(* CODESYS project Tc3_Mc3Ptp.library
   TcLibraryId: Beckhoff Automation GmbH|Tc3_Mc3Ptp|0.4.47.0
   Company: Beckhoff Automation GmbH
   Title: Tc3_Mc3Ptp
   Placeholder: Tc3_Mc3Ptp
   Version: 0.4.47.0

Project tree, tasks and I/O mapping:
  libraries: Tc3_Mc3Base, 0.4.47.0 (Beckhoff Automation GmbH)
  DUTs/
    function block AXIS_REF [ST]: FB_init, FB_exit, InitializeWithOid, GetMotionObjectOid, GetSetValue1DOid, GetActValue1DOid, Name, Oid
    data type AXIS_REF_TOMC
    data type AXIS_REF_TOPLC
    data type EJogMode
    data type EModuloDirection
    Enums/
      data type ELockingStrategy
      data type ETouchProbeSource
    data type EHomingMode
    data type ESource
    data type GearInLegacyOptions
    data type GearInOptions
    data type GearInPosOptions
    data type GearInPosLegacyOptions
    data type SetPositionOptions
    interface Type_ActValue1D: GetActValue1DOid
    interface Type_SetValue1D: GetSetValue1DOid
  POUs/
    Administrative/
      function block MC_Power [ST]: FB_init, FB_exit
      function block MC_SetOverride [ST]: FB_init, FB_exit
      function block MC_Reset [ST]: FB_init, FB_exit
      function block MC_ActivateExternalSetpointGeneration [ST]: FB_init, FB_exit
      function block MC_ReadActualPosition [ST]: FB_init, FB_exit
      function block MC_ReadAxisError [ST]: FB_init, FB_exit
      function block MC_ReadStatus [ST]: FB_init, FB_exit
      function block MC_SetPosition [ST]: FB_init, FB_exit
      function block MC_GetTimeAtActualPosition [ST]: FB_init, FB_exit
      function block MC_GetActualPositionAtTime [ST]: FB_init, FB_exit
      function block MC_TouchProbe [ST]: FB_init, FB_exit
      function block MC_TouchProbeContinuous [ST]: FB_init, FB_exit
      function block MC_AbortTrigger [ST]: FB_init, FB_exit
      function block MC_WriteHardwareParameterAsync [ST]: FB_init, FB_exit
      function block MC_ReadHardwareParameterAsync [ST]: FB_init, FB_exit
    Motion/
      function block MC_Halt [ST]: FB_init, FB_exit
      function block MC_GearIn [ST]: FB_init, FB_exit
      function block MC_GearInLegacy [ST]: FB_init, FB_exit
      function block MC_GearInPos [ST]: FB_init, FB_exit
      function block MC_GearInPosLegacy [ST]: FB_init, FB_exit
      function block MC_MoveAbsolute [ST]: FB_init, FB_exit
      function block MC_MoveModulo [ST]: FB_init, FB_exit
      function block MC_MoveRelative [ST]: FB_init, FB_exit
      function block MC_MoveVelocity [ST]: FB_init, FB_exit
      function block MC_Stop [ST]: FB_init, FB_exit
      function block MC_Home [ST]: FB_init, FB_exit
      function block MC_Jog [ST]: FB_init, FB_exit
      function block MC_WaitForStableActualPosition [ST]: FB_init, FB_exit
      function block MC_PhasingAbsolute [ST]: FB_init, FB_exit
      function block MC_PhasingRelative [ST]: FB_init, FB_exit
      function block MC_HaltPhasing [ST]: FB_init, FB_exit
  Version/
    global variables Global_Version
*)

// DUTs/AXIS_REF_TOMC
(* Contains the information of the AXIS_REF passed from PLC to MC. *)
{attribute 'TcIecLibraryType'}
{attribute 'Namespace' := 'Tc3_Mc3Ptp'}
TYPE AXIS_REF_TOMC : 
	STRUCT
		(* Standard data from PLC to MC. *)
		{attribute 'GUID' := '5A944F05-2D7C-4FD6-9ABA-134068F48E38'}
		{attribute 'Namespace' := 'MC'}
		Std : MC.CDT_PLCTOMC_AXIS_STD;
	END_STRUCT
END_TYPE

// DUTs/AXIS_REF_TOPLC
(* Contains the information of the AXIS_REF passed from PLC to MC. *)
{attribute 'TcIecLibraryType'}
{attribute 'Namespace' := 'Tc3_Mc3Ptp'}
TYPE AXIS_REF_TOPLC : 
	STRUCT
		(* Reference to standard data from MC to PLC. *)
		{attribute 'TcPointerMapping'}
		{attribute 'GUID' := '1FDF4C99-95D5-41A1-806D-90D273DC6BDC'}
		{attribute 'Namespace' := 'MC'}
		Std : REFERENCE TO MC.CDT_MCTOPLC_AXIS_STD;
		(* Reference to setpoint data from MC *)
		{attribute 'TcPointerMapping'}
		{attribute 'GUID' := '619A0C74-EA7E-46BA-B447-F4E8C97E41FB'}
		{attribute 'Namespace' := 'MC'}
		Set : REFERENCE TO MC.CDT_MCTOPLC_AXIS_SET;
		(* Reference to actpoint data from MC *)
		{attribute 'TcPointerMapping'}
		{attribute 'GUID' := 'A42D1F82-D46F-4C1C-8CEF-A7CF7DED130F'}
		{attribute 'Namespace' := 'MC'}
		Act : REFERENCE TO MC.CDT_MCTOPLC_AXIS_ACT;
		 {attribute 'hide'}
		_reserved1 : ARRAY [1..4] OF UINT_8_16;
		(* Reference to modulo positions of a modulo axis *)
		{attribute 'TcPointerMapping'}
		{attribute 'GUID' := 'D0D202B0-695B-4EBE-A25A-AE633C79AA06'}
		{attribute 'Namespace' := 'MC'}
		Modulo : REFERENCE TO MC.CDT_MCTOPLC_AXIS_MODULO;
		(* Reference to load data from MC *)
		{attribute 'TcPointerMapping'}
		{attribute 'GUID' := '222F7CA1-43FF-474A-AC84-1035F5DA7F7A'}
		{attribute 'Namespace' := 'MC'}
		Load : REFERENCE TO MC.CDT_MCTOPLC_AXIS_LOAD;
		 {attribute 'hide'}
		_reserved2 : ARRAY [1..8] OF UINT_8_16;
		(* Reference to fluidpower data from MC *)
		{attribute 'TcPointerMapping'}
		{attribute 'GUID' := 'FF85C83C-7A68-4103-B383-EFF835275DAB'}
		{attribute 'Namespace' := 'MC'}
		FluidPower : REFERENCE TO MC.CDT_MCTOPLC_AXIS_FLUIDPOWER;
	END_STRUCT
END_TYPE

// DUTs/EJogMode
{attribute 'TcIecLibraryType'}
{attribute 'Namespace' := 'Tc3_Mc3Ptp'}
{attribute 'strict'}
{attribute 'qualified_only'}
{attribute 'to_string'}
TYPE EJogMode : (StandardSlow:=1, StandardFast:=2, Continuous:=3, Inching:=4) UINT;
END_TYPE

// DUTs/EModuloDirection
{attribute 'TcIecLibraryType'}
{attribute 'Namespace' := 'Tc3_Mc3Ptp'}
{attribute 'strict'}
{attribute 'qualified_only'}
{attribute 'to_string'}
TYPE EModuloDirection : (ShortestDistance:=0, PositiveDirection:=1, NegativeDirection:=2) UINT;
END_TYPE

// DUTs/EHomingMode
{attribute 'TcIecLibraryType'}
{attribute 'Namespace' := 'Tc3_Mc3Ptp'}
{attribute 'qualified_only'}
{attribute 'strict'}
{attribute 'to_string'}
TYPE EHomingMode : (ForceIsPositionValid:=16#0, ResetIsPositionValid:=16#1, DirectSetPosition:=16#2) UDINT;
END_TYPE

// DUTs/ESource
{attribute 'TcIecLibraryType'}
{attribute 'Namespace' := 'Tc3_Mc3Ptp'}
{attribute 'hide'}
{attribute 'to_string'}
TYPE ESource : (SetValue:=0, ActualValue:=1) UINT;
END_TYPE

// DUTs/GearInLegacyOptions
(* Contains additional options for MC_GearInLegacy *)
{attribute 'TcIecLibraryType'}
{attribute 'Namespace' := 'Tc3_Mc3Ptp'}
{attribute 'hide'}
TYPE GearInLegacyOptions : 
	STRUCT
		{attribute 'Namespace' := 'Tc3_Mc3Base'}
		AllowedSlaveSyncDirections : Tc3_Mc3Base.ESyncDirection := Tc3_Mc3Base.ESyncDirection.Both;
		{attribute 'GUID' := 'AAA4D297-4BFA-4B3F-8507-5BB1F7885E81'}
		{attribute 'Namespace' := 'Tc3_Mc3Ptp'}
		LockingStrategy : ELockingStrategy := ELockingStrategy.PositionLocking;
	END_STRUCT
END_TYPE

// DUTs/GearInOptions
(* Contains additional options for MC_GearIn *)
{attribute 'TcIecLibraryType'}
{attribute 'Namespace' := 'Tc3_Mc3Ptp'}
{attribute 'hide'}
TYPE GearInOptions : 
	STRUCT
		HardcopyWhenInSync : BOOL := false;
	END_STRUCT
END_TYPE

// DUTs/GearInPosOptions
(* Contains additional options for MC_GearInPos *)
{attribute 'TcIecLibraryType'}
{attribute 'Namespace' := 'Tc3_Mc3Ptp'}
{attribute 'hide'}
TYPE GearInPosOptions : 
	STRUCT
		{attribute 'Namespace' := 'Tc3_Mc3Base'}
		AllowedSlaveSyncDirections : Tc3_Mc3Base.ESyncDirection := Tc3_Mc3Base.ESyncDirection.Both;
		 {attribute 'hide'}
		_reserved1 : UINT;
		(* Additional turns for this command *)
		AdditionalTurns : UDINT := 0;
		InSyncToleranceDistance : LREAL := 0;
	END_STRUCT
END_TYPE

// DUTs/GearInPosLegacyOptions
(* Contains additional options for MC_GearInPosLegacy *)
{attribute 'TcIecLibraryType'}
{attribute 'Namespace' := 'Tc3_Mc3Ptp'}
{attribute 'hide'}
TYPE GearInPosLegacyOptions : 
	STRUCT
		{attribute 'Namespace' := 'Tc3_Mc3Base'}
		AllowedSlaveSyncDirections : Tc3_Mc3Base.ESyncDirection := Tc3_Mc3Base.ESyncDirection.Both;
		 {attribute 'hide'}
		_reserved1 : ARRAY [1..6] OF USINT;
		InSyncToleranceDistance : LREAL := 0;
	END_STRUCT
END_TYPE

// DUTs/SetPositionOptions
(* Contains additional options for MC_SetPosition *)
{attribute 'TcIecLibraryType'}
{attribute 'Namespace' := 'Tc3_Mc3Ptp'}
TYPE SetPositionOptions : 
	STRUCT
		(* If TRUE, the position lag is cleared when the function block is executed. *)
		ClearPositionLag : BOOL := false;
	END_STRUCT
END_TYPE

// DUTs/Enums/ELockingStrategy
{attribute 'TcIecLibraryType'}
{attribute 'Namespace' := 'Tc3_Mc3Ptp'}
{attribute 'qualified_only'}
{attribute 'strict'}
{attribute 'to_string'}
TYPE ELockingStrategy : (VelocityLocking:=1, PositionLocking:=2) UINT := VelocityLocking;
END_TYPE

// DUTs/Enums/ETouchProbeSource
(* Selection for touch probe trigger input. *)
{attribute 'TcIecLibraryType'}
{attribute 'Namespace' := 'Tc3_Mc3Ptp'}
{attribute 'qualified_only'}
{attribute 'strict'}
{attribute 'to_string'}
TYPE ETouchProbeSource : (TouchProbe1:=1, TouchProbe2:=2, ExternalTrigger:=3) UINT;
END_TYPE

// Version/Global_Version
{attribute 'TcGenerated'}
// This function has been automatically generated from the project information.
VAR_GLOBAL CONSTANT
	{attribute 'const_non_replaced'}
	{attribute 'linkalways'}
	stLibVersion_Tc3_Mc3Ptp : ST_LibVersion := (iMajor := 0, iMinor := 4, iBuild := 47, iRevision := 0, nFlags := 0, sVersion := '0.4.47.0');
	{attribute 'const_non_replaced'}
	{attribute 'linkalways'}
	sLibraryId_Tc3_Mc3Ptp : String := 'Beckhoff Automation GmbH|Tc3_Mc3Ptp|0.4.47.0';
END_VAR

// DUTs/AXIS_REF

{attribute 'c++_compatible'}
{attribute 'external_name' := 'AXIS_REF_GUID_D3CA51BE_3DF9_1ECF_B7F2_294D2474676B'}
{attribute 'TcIecLibraryType'}
(* AXIS_REF data structure *)
FUNCTION_BLOCK AXIS_REF IMPLEMENTS Tc3_Mc3Base.Type_MotionObject, Type_SetValue1D, Type_ActValue1D
VAR
END_VAR
VAR_INPUT
	(* AXIS_REF outputs. *)
	{attribute 'GUID' := '90A3EB19-687D-4532-BDEE-19D8EA71F7B6'}
	{attribute 'Namespace' := 'Tc3_Mc3Ptp'}
	PlcToMc AT %Q* : AXIS_REF_TOMC;
	(* AXIS_REF inputs. *)
	{attribute 'GUID' := '6F07441C-203E-413F-A1C8-211D3A777892'}
	{attribute 'Namespace' := 'Tc3_Mc3Ptp'}
	McToPlc AT %I* : AXIS_REF_TOPLC;
END_VAR
VAR
	 {attribute 'hide'}
	_reserved1 : ARRAY [1..4] OF UINT_8_16;
END_VAR

{attribute 'TcTypeSystem'}

(* Internal method *)
{attribute 'hide'}
METHOD FB_init : BOOL
VAR_INPUT
	(*  if TRUE, the retain variables are initialized (warm start / cold start) *)
	bInitRetains : BOOL;
	(*  if TRUE, the instance afterwards gets moved into the copy code (online change) *)
	bInCopyCode : BOOL;
END_VAR
END_METHOD

{attribute 'TcTypeSystem'}

(* Internal method *)
{attribute 'hide'}
METHOD FB_exit : BOOL
VAR_INPUT
	(*  if TRUE, the exit method is called for exiting an instance that is copied afterwards (online change). *)
	bInCopyCode : BOOL;
END_VAR
END_METHOD

{attribute 'TcTypeSystem'}

(* Internal method to wrap OID *)
{attribute 'hide'}
METHOD InitializeWithOid
VAR_INPUT
	(*  Oid which is used as an alternative when this is used as master. *)
	{attribute 'GUID' := '18071995-0000-0000-0000-00000000000F'}
	NewOid : GLOBAL.OTCID;
END_VAR
END_METHOD

{attribute 'TcTypeSystem'}

{attribute 'c++_external'}
{attribute 'hide'}
METHOD GetMotionObjectOid : GLOBAL.OTCID
END_METHOD

{attribute 'TcTypeSystem'}

{attribute 'c++_external'}
{attribute 'hide'}
METHOD GetSetValue1DOid : GLOBAL.OTCID
END_METHOD

{attribute 'TcTypeSystem'}

{attribute 'c++_external'}
{attribute 'hide'}
METHOD GetActValue1DOid : GLOBAL.OTCID
END_METHOD

{attribute 'TcTypeSystem'}

{attribute 'monitoring' := 'call'}
	PROPERTY Name : STRING(255)
GET
END_GET
END_PROPERTY

{attribute 'TcTypeSystem'}

{attribute 'monitoring' := 'call'}
	PROPERTY Oid : GLOBAL.OTCID
GET
END_GET
END_PROPERTY

END_FUNCTION_BLOCK

// DUTs/Type_SetValue1D
{attribute 'Namespace' := 'Tc3_Mc3Ptp'}
{attribute 'c++_compatible'}
INTERFACE Type_SetValue1D

{attribute 'TcTypeSystem'}
{attribute 'c++_compatible'}
{attribute 'minimal_input_size' := '4'}
{attribute 'pack_mode' := '4'}
{attribute 'hide'}
METHOD GetSetValue1DOid : GLOBAL.OTCID
END_METHOD

END_INTERFACE

// DUTs/Type_ActValue1D
{attribute 'Namespace' := 'Tc3_Mc3Ptp'}
{attribute 'c++_compatible'}
INTERFACE Type_ActValue1D

{attribute 'TcTypeSystem'}
{attribute 'c++_compatible'}
{attribute 'minimal_input_size' := '4'}
{attribute 'pack_mode' := '4'}
{attribute 'hide'}
METHOD GetActValue1DOid : GLOBAL.OTCID
END_METHOD

END_INTERFACE

// POUs/Administrative/MC_Power

{attribute 'c++_compatible'}
{attribute 'external_name' := 'MC_Power_GUID_E3529116_274C_1460_937E_8AA859633871'}
{attribute 'TcIecLibraryType'}
{attribute 'hide_all_locals'}
(* 
		This function block controls the power stage (on or off).
	 *)
FUNCTION_BLOCK MC_Power
VAR_IN_OUT
	(* Reference to the axis *)
	{attribute 'GUID' := 'D3CA51BE-3DF9-1ECF-B7F2-294D2474676B'}
	{attribute 'Namespace' := 'Tc3_Mc3Ptp'}
	Axis : AXIS_REF;
END_VAR
VAR_INPUT
	(* General software enable for the axis *)
	Enable : BOOL;
	(* Feed enable in positive direction. Only effective if Enable = TRUE *)
	EnablePositive : BOOL := FALSE;
	(* Feed enable in negative direction. Only effective if Enable = TRUE *)
	EnableNegative : BOOL := FALSE;
END_VAR
VAR_OUTPUT
	(* Axis is operationally ready *)
	Status : BOOL;
	(* Axis has error *)
	Error : BOOL;
END_VAR
VAR
	 {attribute 'hide'}
	_reserved1 : ARRAY [1..3] OF USINT;
END_VAR
VAR_OUTPUT
	(* Axis error identifier *)
	ErrorId : UDINT;
END_VAR
VAR
	 {attribute 'hide'}
	_reserved2 : UINT_0_32;
END_VAR

{attribute 'TcTypeSystem'}

(* Internal method *)
{attribute 'hide'}
METHOD FB_init : BOOL
VAR_INPUT
	(*  if TRUE, the retain variables are initialized (warm start / cold start) *)
	bInitRetains : BOOL;
	(*  if TRUE, the instance afterwards gets moved into the copy code (online change) *)
	bInCopyCode : BOOL;
END_VAR
END_METHOD

{attribute 'TcTypeSystem'}

(* Internal method *)
{attribute 'hide'}
METHOD FB_exit : BOOL
VAR_INPUT
	(*  if TRUE, the exit method is called for exiting an instance that is copied afterwards (online change). *)
	bInCopyCode : BOOL;
END_VAR
END_METHOD

END_FUNCTION_BLOCK

// POUs/Administrative/MC_SetOverride

{attribute 'c++_compatible'}
{attribute 'external_name' := 'MC_SetOverride_GUID_121C7E78_08E0_1E5A_A94C_0DF92BBB78C9'}
{attribute 'TcIecLibraryType'}
{attribute 'hide_all_locals'}
(* 
	This function block sets the velocity override factor that is applied to movement commands of the axis.
	The override factor does not apply to movement in the synchronized motion state (e.g. movement induced by MC_GearIn, MC_GearInPos, ...).
	 *)
FUNCTION_BLOCK MC_SetOverride
VAR_IN_OUT
	(* Reference to the axis *)
	{attribute 'GUID' := 'D3CA51BE-3DF9-1ECF-B7F2-294D2474676B'}
	{attribute 'Namespace' := 'Tc3_Mc3Ptp'}
	Axis : AXIS_REF;
END_VAR
VAR_INPUT
	(* Write the velocity override factor continuously while Enable = TRUE *)
	Enable : BOOL;
END_VAR
VAR
	 {attribute 'hide'}
	_reserved1 : ARRAY [1..7] OF USINT;
END_VAR
VAR_INPUT
	(* Applies to commanded velocities. Valid range is [0,1]. Use STRING_TO_LREAL('#Ignore') to NOT overwrite the previous value. *)
	VelocityFactor : LREAL := 1.0;
END_VAR
VAR
	 {attribute 'hide'}
	_reserved2 : ARRAY [1..8] OF USINT;
END_VAR
VAR_OUTPUT
	(* The commanded override is set *)
	Enabled : BOOL;
	(* Error occurred within function block *)
	Error : BOOL;
END_VAR
VAR
	 {attribute 'hide'}
	_reserved3 : UINT;
END_VAR
VAR_OUTPUT
	(* Error identifier *)
	ErrorId : UDINT;
END_VAR

{attribute 'TcTypeSystem'}

(* Internal method *)
{attribute 'hide'}
METHOD FB_init : BOOL
VAR_INPUT
	(*  if TRUE, the retain variables are initialized (warm start / cold start) *)
	bInitRetains : BOOL;
	(*  if TRUE, the instance afterwards gets moved into the copy code (online change) *)
	bInCopyCode : BOOL;
END_VAR
END_METHOD

{attribute 'TcTypeSystem'}

(* Internal method *)
{attribute 'hide'}
METHOD FB_exit : BOOL
VAR_INPUT
	(*  if TRUE, the exit method is called for exiting an instance that is copied afterwards (online change). *)
	bInCopyCode : BOOL;
END_VAR
END_METHOD

END_FUNCTION_BLOCK

// POUs/Motion/MC_GearIn

{attribute 'c++_compatible'}
{attribute 'external_name' := 'MC_GearIn_GUID_E9493D77_974B_13E8_841A_4F997893F8D6'}
{attribute 'TcIecLibraryType'}
{attribute 'hide_all_locals'}
{attribute 'hide'}
(* 
		This function block commands a ratio between the velocity of the slave and master axis.
	 *)
FUNCTION_BLOCK MC_GearIn
VAR_INPUT
	(* Reference to the master axis *)
	{attribute 'GUID' := '67A81BB4-B31C-4E6F-99E0-6B37521E2266'}
	{attribute 'Namespace' := 'Tc3_Mc3Ptp'}
	Master : Type_ActValue1D;
	(* Reference to the slave axis *)
	{attribute 'GUID' := '71DDD02B-B842-4DDB-8CBB-D377B6714EDA'}
	{attribute 'Namespace' := 'Tc3_Mc3Ptp'}
	Slave : Type_SetValue1D;
	(* Trigger the command with rising edge *)
	Execute : BOOL;
END_VAR
VAR
	 {attribute 'hide'}
	_reserved1 : UINT_24_56;
END_VAR
VAR_INPUT
	(* Gear ratio numerator *)
	RatioNumerator : LREAL := 1.0;
	(* Gear ratio denominator *)
	RatioDenominator : UDINT := 1;
END_VAR
VAR
	 {attribute 'hide'}
	_reserved2 : UDINT;
END_VAR
VAR_INPUT
	(* Maximum slave velocity ([PosUnit]/s, positive) *)
	Velocity : LREAL := STRING_TO_LREAL('#Maximum');
	(* Maximum slave acceleration ([PosUnit]/s^2, positive) *)
	Acceleration : LREAL := STRING_TO_LREAL('#Default');
	(* Maximum slave deceleration ([PosUnit]/s^2, positive) *)
	Deceleration : LREAL := STRING_TO_LREAL('#Default');
	(* Maximum slave jerk ([PosUnit]/s^3, positive) *)
	Jerk : LREAL := STRING_TO_LREAL('#Default');
	(* Chronological sequence of the command *)
	{attribute 'Namespace' := 'Tc3_Mc3Base'}
	BufferMode : Tc3_Mc3Base.EBufferMode := Tc3_Mc3Base.EBufferMode.Aborting;
	(* Reaction if an error occurs in the master while this command is active *)
	{attribute 'Namespace' := 'Tc3_Mc3Base'}
	ReactionToMasterError : Tc3_Mc3Base.EReactionToMasterError := Tc3_Mc3Base.EReactionToMasterError.TriggerSlaveError;
	(* Reaction if an error occurs in the slave while this command is active *)
	{attribute 'Namespace' := 'Tc3_Mc3Base'}
	ReactionToSlaveError : Tc3_Mc3Base.EReactionToSlaveError := Tc3_Mc3Base.EReactionToSlaveError.TriggerMasterError;
	(* Advanced function block options *)
	{attribute 'hide'}
	{attribute 'GUID' := 'BA63A6CC-1764-4B99-91C8-CC6CC375B652'}
	{attribute 'Namespace' := 'Tc3_Mc3Ptp'}
	Options : GearInOptions;
END_VAR
VAR_OUTPUT
	(* Synchronization established *)
	InGear : BOOL;
	(* Function block is not finished and new output values are to be expected *)
	Busy : BOOL;
	(* Function block has active control on the axis *)
	Active : BOOL;
	(* Command is aborted by another command *)
	CommandAborted : BOOL;
	(* Error occurred within function block *)
	Error : BOOL;
	(* Error identifier *)
	ErrorId : UDINT;
	(* Master is in error state *)
	MasterHasError : BOOL;
END_VAR
VAR
	 {attribute 'hide'}
	_reserved3 : UINT_24_56;
	 {attribute 'hide'}
	_reserved4 : ARRAY [1..28] OF UINT_8_16;
	 {attribute 'hide'}
	_reserved5 : ARRAY [1..32] OF USINT;
END_VAR

{attribute 'TcTypeSystem'}

(* Internal method *)
{attribute 'hide'}
METHOD FB_init : BOOL
VAR_INPUT
	(*  if TRUE, the retain variables are initialized (warm start / cold start) *)
	bInitRetains : BOOL;
	(*  if TRUE, the instance afterwards gets moved into the copy code (online change) *)
	bInCopyCode : BOOL;
END_VAR
END_METHOD

{attribute 'TcTypeSystem'}

(* Internal method *)
{attribute 'hide'}
METHOD FB_exit : BOOL
VAR_INPUT
	(*  if TRUE, the exit method is called for exiting an instance that is copied afterwards (online change). *)
	bInCopyCode : BOOL;
END_VAR
END_METHOD

END_FUNCTION_BLOCK

// POUs/Motion/MC_GearInPos

{attribute 'c++_compatible'}
{attribute 'external_name' := 'MC_GearInPos_GUID_B2BB4DF7_3ADC_10B7_8213_E2CF5BFD21E3'}
{attribute 'TcIecLibraryType'}
{attribute 'hide_all_locals'}
{attribute 'hide'}
(* 
		This function block commands a gear ratio between the position of the slave and master axes
		from the synchronization point onwards.
	 *)
FUNCTION_BLOCK MC_GearInPos
VAR_INPUT
	(* Reference to the master axis *)
	{attribute 'GUID' := '67A81BB4-B31C-4E6F-99E0-6B37521E2266'}
	{attribute 'Namespace' := 'Tc3_Mc3Ptp'}
	Master : Type_ActValue1D;
	(* Reference to the slave axis *)
	{attribute 'GUID' := '71DDD02B-B842-4DDB-8CBB-D377B6714EDA'}
	{attribute 'Namespace' := 'Tc3_Mc3Ptp'}
	Slave : Type_SetValue1D;
	(* Trigger the command with rising edge *)
	Execute : BOOL;
END_VAR
VAR
	 {attribute 'hide'}
	_reserved1 : UINT_24_56;
END_VAR
VAR_INPUT
	(* Gear ratio numerator *)
	RatioNumerator : LREAL := 1.0;
	(* Gear ratio denominator *)
	RatioDenominator : UDINT := 1;
END_VAR
VAR
	 {attribute 'hide'}
	_reserved2 : UDINT;
END_VAR
VAR_INPUT
	(* Position of master axis where master and slave axis are synchronized *)
	MasterSyncPosition : LREAL := STRING_TO_LREAL('#Invalid');
	(* Position of slave axis where master and slave axis are synchronized *)
	SlaveSyncPosition : LREAL := STRING_TO_LREAL('#Invalid');
	(* Maximum velocity during synchronization ([PosUnit]/s, positive) *)
	Velocity : LREAL := STRING_TO_LREAL('#Maximum');
	(* Maximum acceleration during synchronization ([PosUnit]/s^2, positive) *)
	Acceleration : LREAL := STRING_TO_LREAL('#Default');
	(* Maximum deceleration during synchronization ([PosUnit]/s^2, positive) *)
	Deceleration : LREAL := STRING_TO_LREAL('#Default');
	(* Maximum jerk during synchronization ([PosUnit]/s^3, positive) *)
	Jerk : LREAL := STRING_TO_LREAL('#Default');
	(* Chronological sequence of the command *)
	{attribute 'Namespace' := 'Tc3_Mc3Base'}
	BufferMode : Tc3_Mc3Base.EBufferMode := Tc3_Mc3Base.EBufferMode.Aborting;
	(* Reaction if an error occurs in the master while this command is active *)
	{attribute 'Namespace' := 'Tc3_Mc3Base'}
	ReactionToMasterError : Tc3_Mc3Base.EReactionToMasterError := Tc3_Mc3Base.EReactionToMasterError.TriggerSlaveError;
	(* Reaction if an error occurs in the slave while this command is active *)
	{attribute 'Namespace' := 'Tc3_Mc3Base'}
	ReactionToSlaveError : Tc3_Mc3Base.EReactionToSlaveError := Tc3_Mc3Base.EReactionToSlaveError.TriggerMasterError;
END_VAR
VAR
	 {attribute 'hide'}
	_reserved3 : UINT;
END_VAR
VAR_INPUT
	(* Advanced function block options *)
	{attribute 'hide'}
	{attribute 'GUID' := 'EB67571F-2653-4A23-A3F5-C429B6BFB18A'}
	{attribute 'Namespace' := 'Tc3_Mc3Ptp'}
	Options : GearInPosOptions;
END_VAR
VAR_OUTPUT
	(* Synchronization started *)
	{attribute 'hide'}
	StartSync : BOOL;
	(* Synchronization established *)
	InSync : BOOL;
	(* Function block is not finished and new output values are to be expected *)
	Busy : BOOL;
	(* Function block has active control on the axis *)
	Active : BOOL;
	(* Command is aborted by another command *)
	CommandAborted : BOOL;
	(* Error occurred within function block *)
	Error : BOOL;
END_VAR
VAR
	 {attribute 'hide'}
	_reserved4 : UINT;
END_VAR
VAR_OUTPUT
	(* Error identifier *)
	ErrorId : UDINT;
	(* Master is in error state *)
	MasterHasError : BOOL;
END_VAR
VAR
	 {attribute 'hide'}
	_reserved5 : UINT_24_56;
	 {attribute 'hide'}
	_reserved6 : ARRAY [1..28] OF UINT_8_16;
	 {attribute 'hide'}
	_reserved7 : ARRAY [1..28] OF USINT;
END_VAR

{attribute 'TcTypeSystem'}

(* Internal method *)
{attribute 'hide'}
METHOD FB_init : BOOL
VAR_INPUT
	(*  if TRUE, the retain variables are initialized (warm start / cold start) *)
	bInitRetains : BOOL;
	(*  if TRUE, the instance afterwards gets moved into the copy code (online change) *)
	bInCopyCode : BOOL;
END_VAR
END_METHOD

{attribute 'TcTypeSystem'}

(* Internal method *)
{attribute 'hide'}
METHOD FB_exit : BOOL
VAR_INPUT
	(*  if TRUE, the exit method is called for exiting an instance that is copied afterwards (online change). *)
	bInCopyCode : BOOL;
END_VAR
END_METHOD

END_FUNCTION_BLOCK

// POUs/Administrative/MC_Reset

{attribute 'c++_compatible'}
{attribute 'external_name' := 'MC_Reset_GUID_394AFEA2_BA6F_1DD1_8FD5_98DB85D7F990'}
{attribute 'TcIecLibraryType'}
{attribute 'hide_all_locals'}
(* 
		This function block resets all axis-related errors and transitions the axis out of state ErrorStop.<br/>
		The resulting state is Disabled, if no Enable is requested for the axis (e.g. via MC_Power).<br/>
		It results in DiscreteMotion, if the axis has a closed control loop and a controlled error reaction is still ongoing.<br/>
		Otherwise, standstill is the resultig state. This function block does not affect the output of motion function block instances.
	 *)
FUNCTION_BLOCK MC_Reset
VAR_INPUT
	(* Reference to the axis *)
	{attribute 'Namespace' := 'Tc3_Mc3Base'}
	Axis : Tc3_Mc3Base.Type_MotionObject;
	(* Trigger the command with rising edge *)
	Execute : BOOL;
END_VAR
VAR_OUTPUT
	(* Standstill state is reached *)
	Done : BOOL;
	(* Function block is not finished and new output values are to be expected *)
	Busy : BOOL;
	(* Error occurred within function block *)
	Error : BOOL;
	(* Error identifier *)
	ErrorId : UDINT;
END_VAR
VAR
	 {attribute 'hide'}
	_reserved1 : UINT_0_32;
	 {attribute 'hide'}
	_reserved2 : ARRAY [1..20] OF UINT_8_16;
	 {attribute 'hide'}
	_reserved3 : ARRAY [1..28] OF USINT;
END_VAR

{attribute 'TcTypeSystem'}

(* Internal method *)
{attribute 'hide'}
METHOD FB_init : BOOL
VAR_INPUT
	(*  if TRUE, the retain variables are initialized (warm start / cold start) *)
	bInitRetains : BOOL;
	(*  if TRUE, the instance afterwards gets moved into the copy code (online change) *)
	bInCopyCode : BOOL;
END_VAR
END_METHOD

{attribute 'TcTypeSystem'}

(* Internal method *)
{attribute 'hide'}
METHOD FB_exit : BOOL
VAR_INPUT
	(*  if TRUE, the exit method is called for exiting an instance that is copied afterwards (online change). *)
	bInCopyCode : BOOL;
END_VAR
END_METHOD

END_FUNCTION_BLOCK

// POUs/Administrative/MC_ActivateExternalSetpointGeneration

{attribute 'c++_compatible'}
{attribute 'external_name' := 'MC_ActivateExternalSetpointGeneration_GUID_3255B2A5_BCDE_1F3F_B215_3D486370678C'}
{attribute 'TcIecLibraryType'}
{attribute 'hide_all_locals'}
(* 
		This function block activates external setpoint generation. 
		Setpoints are generated by a function block, which is called through the ITcMcExternalSetpointGenerator interface from the MC context.
		Additionally custom startup data can be passed through the generator.
	 *)
FUNCTION_BLOCK MC_ActivateExternalSetpointGeneration
VAR_INPUT
	(* Reference to the axis *)
	{attribute 'GUID' := '71DDD02B-B842-4DDB-8CBB-D377B6714EDA'}
	{attribute 'Namespace' := 'Tc3_Mc3Ptp'}
	Axis : Type_SetValue1D;
	(* Trigger the command with rising edge *)
	Execute : BOOL;
END_VAR
VAR
	 {attribute 'hide'}
	_reserved1 : UINT_24_56;
END_VAR
VAR_INPUT
	(* External setpoint generator function block *)
	{attribute 'GUID' := 'EF828E0B-69F0-4553-9DFF-4817D2FD6510'}
	ExternalSetpointGenerator : GLOBAL.ITcMcExternalSetpointGenerator;
	(* (reserved) *)
	AllowOtherContext : BOOL := FALSE;
	(* Trigger error on inconsistent setpoint values (position, velocity, acceleration) if EnableDynamicChecks = TRUE *)
	EnableDynamicChecks : BOOL := TRUE;
END_VAR
VAR
	 {attribute 'hide'}
	_reserved2 : UINT_16_48;
END_VAR
VAR_INPUT
	(* Invocation identifier. The InvokeId can be used to identify an external setpoint generator in case external 
		setpoint generation is activated multiple times with the same ExternalSetpointGenerator. Another possibility is to transfer 
		custom data (for example a pointer to data struct) by this InvokeId. *)
	{attribute 'GUID' := '18071995-0000-0000-0000-000000000073'}
	{attribute 'GlobalType'}
	InvokeId : GLOBAL.XWORD := 0;
	(* Chronological sequence of the command *)
	{attribute 'Namespace' := 'Tc3_Mc3Base'}
	BufferMode : Tc3_Mc3Base.EBufferMode := Tc3_Mc3Base.EBufferMode.Aborting;
END_VAR
VAR_OUTPUT
	(* Function block is not finished and new output values are to be expected *)
	Busy : BOOL;
	(* Function block has active control on the axis *)
	Active : BOOL;
	(* Command is aborted by another command *)
	CommandAborted : BOOL;
	(* Error occurred within function block *)
	Error : BOOL;
END_VAR
VAR
	 {attribute 'hide'}
	_reserved3 : UINT;
END_VAR
VAR_OUTPUT
	(* Error identifier *)
	ErrorId : UDINT;
END_VAR
VAR
	 {attribute 'hide'}
	_reserved4 : UINT_0_32;
	 {attribute 'hide'}
	_reserved5 : ARRAY [1..32] OF UINT_8_16;
	 {attribute 'hide'}
	_reserved6 : ARRAY [1..24] OF USINT;
END_VAR

{attribute 'TcTypeSystem'}

(* Internal method *)
{attribute 'hide'}
METHOD FB_init : BOOL
VAR_INPUT
	(*  if TRUE, the retain variables are initialized (warm start / cold start) *)
	bInitRetains : BOOL;
	(*  if TRUE, the instance afterwards gets moved into the copy code (online change) *)
	bInCopyCode : BOOL;
END_VAR
END_METHOD

{attribute 'TcTypeSystem'}

(* Internal method *)
{attribute 'hide'}
METHOD FB_exit : BOOL
VAR_INPUT
	(*  if TRUE, the exit method is called for exiting an instance that is copied afterwards (online change). *)
	bInCopyCode : BOOL;
END_VAR
END_METHOD

END_FUNCTION_BLOCK

// POUs/Administrative/MC_ReadActualPosition

{attribute 'c++_compatible'}
{attribute 'external_name' := 'MC_ReadActualPosition_GUID_3C39B8D5_BF98_1B0D_873D_11943FFCDFE9'}
{attribute 'TcIecLibraryType'}
{attribute 'hide_all_locals'}
{attribute 'hide'}
(* 
		This function block reads the current axis actual position.
	 *)
FUNCTION_BLOCK MC_ReadActualPosition
VAR_IN_OUT
	(* Reference to the axis *)
	{attribute 'GUID' := 'D3CA51BE-3DF9-1ECF-B7F2-294D2474676B'}
	{attribute 'Namespace' := 'Tc3_Mc3Ptp'}
	Axis : AXIS_REF;
END_VAR
VAR_INPUT
	(* Read the actual position continuously while Enable = TRUE *)
	Enable : BOOL;
END_VAR
VAR_OUTPUT
	(* Valid output available at function block *)
	Valid : BOOL;
	(* Function block is not finished and new output values are to be expected *)
	Busy : BOOL;
	(* Error occurred within function block *)
	Error : BOOL;
	(* Error identifier *)
	ErrorId : UDINT;
	(* Actual position ([PosUnit]) *)
	Position : LREAL;
END_VAR

{attribute 'TcTypeSystem'}

(* Internal method *)
{attribute 'hide'}
METHOD FB_init : BOOL
VAR_INPUT
	(*  if TRUE, the retain variables are initialized (warm start / cold start) *)
	bInitRetains : BOOL;
	(*  if TRUE, the instance afterwards gets moved into the copy code (online change) *)
	bInCopyCode : BOOL;
END_VAR
END_METHOD

{attribute 'TcTypeSystem'}

(* Internal method *)
{attribute 'hide'}
METHOD FB_exit : BOOL
VAR_INPUT
	(*  if TRUE, the exit method is called for exiting an instance that is copied afterwards (online change). *)
	bInCopyCode : BOOL;
END_VAR
END_METHOD

END_FUNCTION_BLOCK

// POUs/Administrative/MC_ReadAxisError

{attribute 'c++_compatible'}
{attribute 'external_name' := 'MC_ReadAxisError_GUID_C6F572C1_61AE_1DA6_A376_F0A2AD8A74DD'}
{attribute 'TcIecLibraryType'}
{attribute 'hide_all_locals'}
{attribute 'hide'}
(* 
		This function block reads the current axis error identifier.
	 *)
FUNCTION_BLOCK MC_ReadAxisError
VAR_IN_OUT
	(* Reference to the axis *)
	{attribute 'GUID' := 'D3CA51BE-3DF9-1ECF-B7F2-294D2474676B'}
	{attribute 'Namespace' := 'Tc3_Mc3Ptp'}
	Axis : AXIS_REF;
END_VAR
VAR_INPUT
	(* Read the axis error identifier continuously while Enable = TRUE *)
	Enable : BOOL;
END_VAR
VAR_OUTPUT
	(* Valid output available at function block *)
	Valid : BOOL;
	(* Function block is not finished and new output values are to be expected *)
	Busy : BOOL;
	(* Error occurred within function block *)
	Error : BOOL;
	(* Error identifier *)
	ErrorId : UDINT;
	(* Axis error identifier *)
	AxisErrorId : UDINT;
END_VAR
VAR
	 {attribute 'hide'}
	_reserved1 : UINT_0_32;
END_VAR

{attribute 'TcTypeSystem'}

(* Internal method *)
{attribute 'hide'}
METHOD FB_init : BOOL
VAR_INPUT
	(*  if TRUE, the retain variables are initialized (warm start / cold start) *)
	bInitRetains : BOOL;
	(*  if TRUE, the instance afterwards gets moved into the copy code (online change) *)
	bInCopyCode : BOOL;
END_VAR
END_METHOD

{attribute 'TcTypeSystem'}

(* Internal method *)
{attribute 'hide'}
METHOD FB_exit : BOOL
VAR_INPUT
	(*  if TRUE, the exit method is called for exiting an instance that is copied afterwards (online change). *)
	bInCopyCode : BOOL;
END_VAR
END_METHOD

END_FUNCTION_BLOCK

// POUs/Administrative/MC_ReadStatus

{attribute 'c++_compatible'}
{attribute 'external_name' := 'MC_ReadStatus_GUID_294643E2_96D8_11B0_8DA0_D7A71A4F8120'}
{attribute 'TcIecLibraryType'}
{attribute 'hide_all_locals'}
(* 
		This function block reads the current axis state.
	 *)
FUNCTION_BLOCK MC_ReadStatus
VAR_IN_OUT
	(* Reference to the axis *)
	{attribute 'GUID' := 'D3CA51BE-3DF9-1ECF-B7F2-294D2474676B'}
	{attribute 'Namespace' := 'Tc3_Mc3Ptp'}
	Axis : AXIS_REF;
END_VAR
VAR_INPUT
	(* Read the axis state continuously while Enable = TRUE *)
	Enable : BOOL;
END_VAR
VAR_OUTPUT
	(* Valid output available at function block *)
	Valid : BOOL;
	(* Error occurred within function block *)
	Error : BOOL;
END_VAR
VAR
	 {attribute 'hide'}
	_reserved1 : USINT;
END_VAR
VAR_OUTPUT
	(* Error identifier *)
	ErrorId : UDINT;
	(* Axis is in state ErrorStop *)
	ErrorStop : BOOL;
	(* Axis is in state Disabled *)
	Disabled : BOOL;
	(* Axis is in state Stopping *)
	Stopping : BOOL;
	(* Axis is in state Homing *)
	Homing : BOOL;
	(* Axis is in state Standstill *)
	Standstill : BOOL;
	(* Axis is in state DiscreteMotion *)
	DiscreteMotion : BOOL;
	(* Axis is in state ContinuousMotion *)
	ContinuousMotion : BOOL;
	(* Axis is in state SynchronizedMotion *)
	SynchronizedMotion : BOOL;
END_VAR

{attribute 'TcTypeSystem'}

(* Internal method *)
{attribute 'hide'}
METHOD FB_init : BOOL
VAR_INPUT
	(*  if TRUE, the retain variables are initialized (warm start / cold start) *)
	bInitRetains : BOOL;
	(*  if TRUE, the instance afterwards gets moved into the copy code (online change) *)
	bInCopyCode : BOOL;
END_VAR
END_METHOD

{attribute 'TcTypeSystem'}

(* Internal method *)
{attribute 'hide'}
METHOD FB_exit : BOOL
VAR_INPUT
	(*  if TRUE, the exit method is called for exiting an instance that is copied afterwards (online change). *)
	bInCopyCode : BOOL;
END_VAR
END_METHOD

END_FUNCTION_BLOCK

// POUs/Administrative/MC_SetPosition

{attribute 'c++_compatible'}
{attribute 'external_name' := 'MC_SetPosition_GUID_75691C58_C510_1BCF_81F5_23E77C57D1A7'}
{attribute 'TcIecLibraryType'}
{attribute 'hide_all_locals'}
(* 
		This function block shifts the coordinate system of an axis by manipulating both the setpoint position as well as the
		actual position of an axis with the same value without any movement caused (Re-calibration with same following error).
		This can be used for instance for a reference situation.
	 *)
FUNCTION_BLOCK MC_SetPosition
VAR_INPUT
	(* Reference to the axis *)
	{attribute 'GUID' := '71DDD02B-B842-4DDB-8CBB-D377B6714EDA'}
	{attribute 'Namespace' := 'Tc3_Mc3Ptp'}
	Axis : Type_SetValue1D;
	(* Trigger the command with rising edge *)
	Execute : BOOL;
END_VAR
VAR
	 {attribute 'hide'}
	_reserved1 : ARRAY [1..7] OF USINT;
END_VAR
VAR_INPUT
	(* New position value ([PosUnit]) or distance if Relative = TRUE *)
	Position : LREAL := STRING_TO_LREAL('#Invalid');
	(* Shift axis position by value *)
	Relative : BOOL := FALSE;
	(* Advanced function block options *)
	{attribute 'GUID' := '8BDBC654-D053-42BE-BD59-268374CF5136'}
	{attribute 'Namespace' := 'Tc3_Mc3Ptp'}
	Options : SetPositionOptions;
END_VAR
VAR_OUTPUT
	(* Position has new value *)
	Done : BOOL;
	(* Function block is not finished and new output values are to be expected *)
	Busy : BOOL;
	(* Error occurred within function block *)
	Error : BOOL;
END_VAR
VAR
	 {attribute 'hide'}
	_reserved2 : ARRAY [1..3] OF USINT;
END_VAR
VAR_OUTPUT
	(* Error identifier *)
	ErrorId : UDINT;
END_VAR
VAR
	 {attribute 'hide'}
	_reserved3 : UINT_0_32;
	 {attribute 'hide'}
	_reserved4 : ARRAY [1..20] OF UINT_8_16;
	 {attribute 'hide'}
	_reserved5 : ARRAY [1..32] OF USINT;
END_VAR

{attribute 'TcTypeSystem'}

(* Internal method *)
{attribute 'hide'}
METHOD FB_init : BOOL
VAR_INPUT
	(*  if TRUE, the retain variables are initialized (warm start / cold start) *)
	bInitRetains : BOOL;
	(*  if TRUE, the instance afterwards gets moved into the copy code (online change) *)
	bInCopyCode : BOOL;
END_VAR
END_METHOD

{attribute 'TcTypeSystem'}

(* Internal method *)
{attribute 'hide'}
METHOD FB_exit : BOOL
VAR_INPUT
	(*  if TRUE, the exit method is called for exiting an instance that is copied afterwards (online change). *)
	bInCopyCode : BOOL;
END_VAR
END_METHOD

END_FUNCTION_BLOCK

// POUs/Administrative/MC_GetTimeAtActualPosition

{attribute 'c++_compatible'}
{attribute 'external_name' := 'MC_GetTimeAtActualPosition_GUID_0CA0D808_4FD4_1C4C_BDA4_507861BABE74'}
{attribute 'TcIecLibraryType'}
{attribute 'hide_all_locals'}
(* 
		This function block determines the DC time for an actual position. 
		The DC time is approximated by an extrapolation based on the current actual position and velocity. 
		An error is triggered if the axis is stationary (velocity = 0.0)
	 *)
FUNCTION_BLOCK MC_GetTimeAtActualPosition
VAR_IN_OUT
	(* Reference to the axis *)
	{attribute 'GUID' := 'D3CA51BE-3DF9-1ECF-B7F2-294D2474676B'}
	{attribute 'Namespace' := 'Tc3_Mc3Ptp'}
	Axis : AXIS_REF;
END_VAR
VAR_INPUT
	(* Get the DC time continuously while Enable = TRUE *)
	Enable : BOOL;
END_VAR
VAR
	 {attribute 'hide'}
	_reserved1 : ARRAY [1..7] OF USINT;
END_VAR
VAR_INPUT
	(* Actual position *)
	Position : LREAL := STRING_TO_LREAL('#Invalid');
END_VAR
VAR_OUTPUT
	(* Valid output available at function block *)
	Valid : BOOL;
	(* Error occurred within function block *)
	Error : BOOL;
END_VAR
VAR
	 {attribute 'hide'}
	_reserved2 : UINT;
END_VAR
VAR_OUTPUT
	(* Error identifier *)
	ErrorId : UDINT;
	(* DC time at requested position *)
	DcTimeAtPosition : LINT;
END_VAR

{attribute 'TcTypeSystem'}

(* Internal method *)
{attribute 'hide'}
METHOD FB_init : BOOL
VAR_INPUT
	(*  if TRUE, the retain variables are initialized (warm start / cold start) *)
	bInitRetains : BOOL;
	(*  if TRUE, the instance afterwards gets moved into the copy code (online change) *)
	bInCopyCode : BOOL;
END_VAR
END_METHOD

{attribute 'TcTypeSystem'}

(* Internal method *)
{attribute 'hide'}
METHOD FB_exit : BOOL
VAR_INPUT
	(*  if TRUE, the exit method is called for exiting an instance that is copied afterwards (online change). *)
	bInCopyCode : BOOL;
END_VAR
END_METHOD

END_FUNCTION_BLOCK

// POUs/Administrative/MC_GetActualPositionAtTime

{attribute 'c++_compatible'}
{attribute 'external_name' := 'MC_GetActualPositionAtTime_GUID_23645428_D10F_19DF_9459_FD3291FE93CB'}
{attribute 'TcIecLibraryType'}
{attribute 'hide_all_locals'}
(* 
		This function block returns the actual position for a DC time. 
		If the DC time value is not within the last 64 MET cycles, the position is approximated by an extrapolation.
	 *)
FUNCTION_BLOCK MC_GetActualPositionAtTime
VAR_INPUT
	(* Reference to the axis *)
	{attribute 'GUID' := '67A81BB4-B31C-4E6F-99E0-6B37521E2266'}
	{attribute 'Namespace' := 'Tc3_Mc3Ptp'}
	Axis : Type_ActValue1D;
	(* Get the actual position continuously while Enable = TRUE *)
	Enable : BOOL;
END_VAR
VAR
	 {attribute 'hide'}
	_reserved1 : ARRAY [1..7] OF USINT;
END_VAR
VAR_INPUT
	(* DC time value *)
	DcTime : LINT := 0;
END_VAR
VAR_OUTPUT
	(* Valid output available at function block *)
	Valid : BOOL;
	(* Error occurred within function block *)
	Error : BOOL;
END_VAR
VAR
	 {attribute 'hide'}
	_reserved2 : UINT;
END_VAR
VAR_OUTPUT
	(* Error identifier *)
	ErrorId : UDINT;
	(* Actual position at requested DC time *)
	PositionAtDcTime : LREAL;
END_VAR

{attribute 'TcTypeSystem'}

(* Internal method *)
{attribute 'hide'}
METHOD FB_init : BOOL
VAR_INPUT
	(*  if TRUE, the retain variables are initialized (warm start / cold start) *)
	bInitRetains : BOOL;
	(*  if TRUE, the instance afterwards gets moved into the copy code (online change) *)
	bInCopyCode : BOOL;
END_VAR
END_METHOD

{attribute 'TcTypeSystem'}

(* Internal method *)
{attribute 'hide'}
METHOD FB_exit : BOOL
VAR_INPUT
	(*  if TRUE, the exit method is called for exiting an instance that is copied afterwards (online change). *)
	bInCopyCode : BOOL;
END_VAR
END_METHOD

END_FUNCTION_BLOCK

// POUs/Administrative/MC_TouchProbe

{attribute 'c++_compatible'}
{attribute 'external_name' := 'MC_TouchProbe_GUID_BCE723C4_D2E1_1BCF_B3F6_8BFEAF54F069'}
{attribute 'TcIecLibraryType'}
{attribute 'hide_all_locals'}
(* 
		This function block controls the recording of an axis position at a trigger event by the drive.<br/>
		After the Execute input is set, the first recorded position / event inside the specified window can be read at the Recorded.. outputs.<br/>
		One of WindowFirstPosition or WindowLastPosition can be left as 'Ignore' if no corresponding limit is desired.
	 *)
FUNCTION_BLOCK MC_TouchProbe
VAR_INPUT
	(* Reference to the axis *)
	{attribute 'GUID' := '67A81BB4-B31C-4E6F-99E0-6B37521E2266'}
	{attribute 'Namespace' := 'Tc3_Mc3Ptp'}
	Axis : Type_ActValue1D;
	(* Trigger the command with rising edge *)
	Execute : BOOL;
END_VAR
VAR
	 {attribute 'hide'}
	_reserved1 : USINT;
END_VAR
VAR_INPUT
	(* Trigger signal source. Valid values: 1 = TouchProbe1, 2 = TouchProbe2, 3 = ExternalTrigger *)
	TriggerSource : UINT := 1;
	(* Edge of trigger signal at which position is recorded. Valid values: 0 = RisingEdge, 1 = FallingEdge *)
	SignalEdgeEvaluation : UINT := 0;
END_VAR
VAR
	 {attribute 'hide'}
	_reserved2 : UINT;
END_VAR
VAR_INPUT
	(* DcTime of trigger event. Must be set if external trigger is used. *)
	DcTime : LINT := 0;
	(* Start position from where trigger events are accepted ([PosUnit], included in the position window).
		It can be left as 'Ignore' if no lower limit is desired. Must have value <= WindowLastPosition otherwise. *)
	WindowFirstPosition : LREAL := STRING_TO_LREAL('#Ignore');
	(* Stop position up to where trigger events are accepted ([PosUnit], included in the position window).
		It can be left as 'Ignore' if no upper limit is desired. Must have value >= WindowFirstPosition otherwise.
		 *)
	WindowLastPosition : LREAL := STRING_TO_LREAL('#Ignore');
	(* Calculate RecordedPosition as modulo value *)
	PositionsAsModuloValues : BOOL := FALSE;
END_VAR
VAR
	 {attribute 'hide'}
	_reserved3 : ARRAY [1..7] OF USINT;
END_VAR
VAR_OUTPUT
	(* Position where trigger event occurred ([PosUnit]) *)
	RecordedPosition : LREAL;
	(* DcTime at trigger event *)
	RecordedDcTime : LINT;
	(* Number of recorded trigger events *)
	{attribute 'hide'}
	Counter : UDINT;
	(* Touch probe process succeeded *)
	Done : BOOL;
	(* Function block is not finished and new output values are to be expected *)
	Busy : BOOL;
END_VAR
VAR
	 {attribute 'hide'}
	_reserved4 : USINT;
END_VAR
VAR_OUTPUT
	(* Command is aborted by another command *)
	CommandAborted : BOOL;
	(* Error occurred within function block *)
	Error : BOOL;
END_VAR
VAR
	 {attribute 'hide'}
	_reserved5 : ARRAY [1..3] OF USINT;
END_VAR
VAR_OUTPUT
	(* Error identifier *)
	ErrorId : UDINT;
END_VAR
VAR
	 {attribute 'hide'}
	_reserved6 : UINT_0_32;
	 {attribute 'hide'}
	_reserved7 : ARRAY [1..28] OF UINT_8_16;
	 {attribute 'hide'}
	_reserved8 : ARRAY [1..36] OF USINT;
END_VAR

{attribute 'TcTypeSystem'}

(* Internal method *)
{attribute 'hide'}
METHOD FB_init : BOOL
VAR_INPUT
	(*  if TRUE, the retain variables are initialized (warm start / cold start) *)
	bInitRetains : BOOL;
	(*  if TRUE, the instance afterwards gets moved into the copy code (online change) *)
	bInCopyCode : BOOL;
END_VAR
END_METHOD

{attribute 'TcTypeSystem'}

(* Internal method *)
{attribute 'hide'}
METHOD FB_exit : BOOL
VAR_INPUT
	(*  if TRUE, the exit method is called for exiting an instance that is copied afterwards (online change). *)
	bInCopyCode : BOOL;
END_VAR
END_METHOD

END_FUNCTION_BLOCK

// POUs/Administrative/MC_TouchProbeContinuous

{attribute 'c++_compatible'}
{attribute 'external_name' := 'MC_TouchProbeContinuous_GUID_1051196C_E9F6_1C36_96C4_F1CD0D12B136'}
{attribute 'TcIecLibraryType'}
{attribute 'hide_all_locals'}
(* 
		This function block controls the recording of an axis position at a trigger event by the drive.<br/>
		While the Enable input is set, recorded positions / events inside the specified window can be read at the Recorded.. outputs.<br/>
		One of WindowFirstPosition or WindowLastPosition can be left as 'Ignore' if no corresponding limit is desired.
	 *)
FUNCTION_BLOCK MC_TouchProbeContinuous
VAR_INPUT
	(* Reference to the axis *)
	{attribute 'GUID' := '67A81BB4-B31C-4E6F-99E0-6B37521E2266'}
	{attribute 'Namespace' := 'Tc3_Mc3Ptp'}
	Axis : Type_ActValue1D;
	(* Run the touch probe process continuously while Enable = TRUE *)
	Enable : BOOL;
END_VAR
VAR
	 {attribute 'hide'}
	_reserved1 : USINT;
END_VAR
VAR_INPUT
	(* Trigger signal source. Valid values: 1 = TouchProbe1, 2 = TouchProbe2, 3 = ExternalTrigger *)
	TriggerSource : UINT := 1;
	(* Edge of trigger signal at which position is recorded. Valid values: 0 = RisingEdge, 1 = FallingEdge *)
	SignalEdgeEvaluation : UINT := 0;
END_VAR
VAR
	 {attribute 'hide'}
	_reserved2 : UINT;
END_VAR
VAR_INPUT
	(* DcTime of trigger event. Must be set if external trigger is used. *)
	DcTime : LINT := 0;
	(* Start position from where (positive direction) trigger events are accepted ([PosUnit], included in the position window).
		It can be left as 'Ignore' if no lower limit is desired. Must have value <= WindowLastPosition otherwise.
		 *)
	WindowFirstPosition : LREAL := STRING_TO_LREAL('#Ignore');
	(* Stop position up to where (positive direction) trigger events are accepted ([PosUnit], included in the position window).
		It can be left as 'Ignore' if no upper limit is desired. Must have value >= WindowFirstPosition otherwise.
		 *)
	WindowLastPosition : LREAL := STRING_TO_LREAL('#Ignore');
	(* Calculate RecordedPosition as modulo value *)
	PositionsAsModuloValues : BOOL := FALSE;
END_VAR
VAR
	 {attribute 'hide'}
	_reserved3 : ARRAY [1..7] OF USINT;
END_VAR
VAR_OUTPUT
	(* Position where trigger event occurred ([PosUnit]) *)
	RecordedPosition : LREAL;
	(* DcTime at trigger event *)
	RecordedDcTime : LINT;
	(* Number of recorded trigger events *)
	{attribute 'hide'}
	Counter : UDINT;
	(* Valid output available at Function Block *)
	Valid : BOOL;
	(* Function block is not finished and new output values are to be expected *)
	Busy : BOOL;
END_VAR
VAR
	 {attribute 'hide'}
	_reserved4 : USINT;
END_VAR
VAR_OUTPUT
	(* Command is aborted by another command *)
	CommandAborted : BOOL;
	(* Error occurred within function block *)
	Error : BOOL;
END_VAR
VAR
	 {attribute 'hide'}
	_reserved5 : ARRAY [1..3] OF USINT;
END_VAR
VAR_OUTPUT
	(* Error identifier *)
	ErrorId : UDINT;
END_VAR
VAR
	 {attribute 'hide'}
	_reserved6 : UINT_0_32;
	 {attribute 'hide'}
	_reserved7 : ARRAY [1..28] OF UINT_8_16;
	 {attribute 'hide'}
	_reserved8 : ARRAY [1..60] OF USINT;
END_VAR

{attribute 'TcTypeSystem'}

(* Internal method *)
{attribute 'hide'}
METHOD FB_init : BOOL
VAR_INPUT
	(*  if TRUE, the retain variables are initialized (warm start / cold start) *)
	bInitRetains : BOOL;
	(*  if TRUE, the instance afterwards gets moved into the copy code (online change) *)
	bInCopyCode : BOOL;
END_VAR
END_METHOD

{attribute 'TcTypeSystem'}

(* Internal method *)
{attribute 'hide'}
METHOD FB_exit : BOOL
VAR_INPUT
	(*  if TRUE, the exit method is called for exiting an instance that is copied afterwards (online change). *)
	bInCopyCode : BOOL;
END_VAR
END_METHOD

END_FUNCTION_BLOCK

// POUs/Administrative/MC_AbortTrigger

{attribute 'c++_compatible'}
{attribute 'external_name' := 'MC_AbortTrigger_GUID_C53A86B5_E909_1B37_B302_EC0809948178'}
{attribute 'TcIecLibraryType'}
{attribute 'hide_all_locals'}
(* 
		This function block is used to abort function blocks which are connected to trigger events (e.g. MC_TouchProbe).
	 *)
FUNCTION_BLOCK MC_AbortTrigger
VAR_INPUT
	(* Reference to the axis *)
	{attribute 'GUID' := '71DDD02B-B842-4DDB-8CBB-D377B6714EDA'}
	{attribute 'Namespace' := 'Tc3_Mc3Ptp'}
	Axis : Type_SetValue1D;
	(* Trigger the command with rising edge *)
	Execute : BOOL;
END_VAR
VAR
	 {attribute 'hide'}
	_reserved1 : USINT;
END_VAR
VAR_INPUT
	(* Trigger signal source. Valid values: 1 = TouchProbe1, 2 = TouchProbe2 *)
	TriggerSource : UINT := 1;
	(* Edge of trigger signal at which position is recorded. Valid values: 0 = RisingEdge, 1 = FallingEdge *)
	SignalEdgeEvaluation : UINT := 0;
END_VAR
VAR_OUTPUT
	(* The recording of touch probe events for the given signal source and signal edge is aborted *)
	Done : BOOL;
	(* Function block is not finished and new output values are to be expected *)
	Busy : BOOL;
	(* Error occurred within function block *)
	Error : BOOL;
END_VAR
VAR
	 {attribute 'hide'}
	_reserved2 : ARRAY [1..3] OF USINT;
END_VAR
VAR_OUTPUT
	(* Error identifier *)
	ErrorId : UDINT;
END_VAR
VAR
	 {attribute 'hide'}
	_reserved3 : UINT_0_32;
	 {attribute 'hide'}
	_reserved4 : ARRAY [1..28] OF UINT_8_16;
	 {attribute 'hide'}
	_reserved5 : ARRAY [1..28] OF USINT;
END_VAR

{attribute 'TcTypeSystem'}

(* Internal method *)
{attribute 'hide'}
METHOD FB_init : BOOL
VAR_INPUT
	(*  if TRUE, the retain variables are initialized (warm start / cold start) *)
	bInitRetains : BOOL;
	(*  if TRUE, the instance afterwards gets moved into the copy code (online change) *)
	bInCopyCode : BOOL;
END_VAR
END_METHOD

{attribute 'TcTypeSystem'}

(* Internal method *)
{attribute 'hide'}
METHOD FB_exit : BOOL
VAR_INPUT
	(*  if TRUE, the exit method is called for exiting an instance that is copied afterwards (online change). *)
	bInCopyCode : BOOL;
END_VAR
END_METHOD

END_FUNCTION_BLOCK

// POUs/Administrative/MC_WriteHardwareParameterAsync

{attribute 'c++_compatible'}
{attribute 'external_name' := 'MC_WriteHardwareParameterAsync_GUID_F23632D0_F3B6_1A1A_9B8A_E0860CB3E8DE'}
{attribute 'TcIecLibraryType'}
{attribute 'hide_all_locals'}
(* 
		This function block writes parameters to the hardware drive.
		It supports CoE and SoE drives.
	 *)
FUNCTION_BLOCK MC_WriteHardwareParameterAsync
VAR_INPUT
	(* Reference to the axis *)
	{attribute 'Namespace' := 'Tc3_Mc3Base'}
	Axis : Tc3_Mc3Base.Type_MotionObject;
	(* Execute *)
	Execute : BOOL;
END_VAR
VAR
	 {attribute 'hide'}
	_reserved1 : USINT;
END_VAR
VAR_INPUT
	(* CoE object index or SoE IDN *)
	Index : UINT := 0;
	(* CoE sub index or SoE element *)
	SubIndex : USINT := 0;
END_VAR
VAR
	 {attribute 'hide'}
	_reserved2 : ARRAY [1..3] OF USINT;
END_VAR
VAR_INPUT
	(* Contains the address of the data. *)
	{attribute 'GUID' := '18071995-0000-0000-0000-000000000018'}
	{attribute 'GlobalType'}
	AddrValue : GLOBAL.PVOID := 0;
	(* Contains the size of the data. *)
	SizeValue : UDINT := 0;
END_VAR
VAR_OUTPUT
	(* Value is successfully sent to the target. *)
	Done : BOOL;
	(* Function block is not finished. *)
	Busy : BOOL;
	(* Function block is active. *)
	Active : BOOL;
	(* Error occurred within function block. *)
	Error : BOOL;
	(* Error identifier *)
	ErrorId : UDINT;
END_VAR
VAR
	 {attribute 'hide'}
	_reserved3 : UINT_0_32;
	 {attribute 'hide'}
	_reserved4 : ARRAY [1..32] OF UINT_8_16;
	 {attribute 'hide'}
	_reserved5 : ARRAY [1..32] OF USINT;
END_VAR

{attribute 'TcTypeSystem'}

(* Internal method *)
{attribute 'hide'}
METHOD FB_init : BOOL
VAR_INPUT
	(*  if TRUE, the retain variables are initialized (warm start / cold start) *)
	bInitRetains : BOOL;
	(*  if TRUE, the instance afterwards gets moved into the copy code (online change) *)
	bInCopyCode : BOOL;
END_VAR
END_METHOD

{attribute 'TcTypeSystem'}

(* Internal method *)
{attribute 'hide'}
METHOD FB_exit : BOOL
VAR_INPUT
	(*  if TRUE, the exit method is called for exiting an instance that is copied afterwards (online change). *)
	bInCopyCode : BOOL;
END_VAR
END_METHOD

END_FUNCTION_BLOCK

// POUs/Administrative/MC_ReadHardwareParameterAsync

{attribute 'c++_compatible'}
{attribute 'external_name' := 'MC_ReadHardwareParameterAsync_GUID_2D9464C1_C289_1B6B_9D2D_C1C10C768F7A'}
{attribute 'TcIecLibraryType'}
{attribute 'hide_all_locals'}
(* 
		This function block reads parameters to the hardware drive. The function block supports CoE and SoE drives.
	 *)
FUNCTION_BLOCK MC_ReadHardwareParameterAsync
VAR_INPUT
	(* Reference to the axis *)
	{attribute 'Namespace' := 'Tc3_Mc3Base'}
	Axis : Tc3_Mc3Base.Type_MotionObject;
	(* Trigger the command with rising edge *)
	Execute : BOOL;
END_VAR
VAR
	 {attribute 'hide'}
	_reserved1 : USINT;
END_VAR
VAR_INPUT
	(* CoE object index or SoE IDN *)
	Index : UINT := 0;
	(* CoE sub index or SoE element *)
	SubIndex : USINT := 0;
END_VAR
VAR
	 {attribute 'hide'}
	_reserved2 : ARRAY [1..3] OF USINT;
END_VAR
VAR_INPUT
	(* Contains the address of the data. *)
	{attribute 'GUID' := '18071995-0000-0000-0000-000000000018'}
	{attribute 'GlobalType'}
	AddrValue : GLOBAL.PVOID := 0;
	(* Contains the size of the data. *)
	SizeValue : UDINT := 0;
END_VAR
VAR_OUTPUT
	(* Value is successfully sent to the target. *)
	Done : BOOL;
	(* Function block is not finished *)
	Busy : BOOL;
	(* Function block is active. *)
	Active : BOOL;
	(* Error occurred within function block *)
	Error : BOOL;
	(* Error identifier *)
	ErrorId : UDINT;
END_VAR
VAR
	 {attribute 'hide'}
	_reserved3 : UINT_0_32;
	 {attribute 'hide'}
	_reserved4 : ARRAY [1..32] OF UINT_8_16;
	 {attribute 'hide'}
	_reserved5 : ARRAY [1..32] OF USINT;
END_VAR

{attribute 'TcTypeSystem'}

(* Internal method *)
{attribute 'hide'}
METHOD FB_init : BOOL
VAR_INPUT
	(*  if TRUE, the retain variables are initialized (warm start / cold start) *)
	bInitRetains : BOOL;
	(*  if TRUE, the instance afterwards gets moved into the copy code (online change) *)
	bInCopyCode : BOOL;
END_VAR
END_METHOD

{attribute 'TcTypeSystem'}

(* Internal method *)
{attribute 'hide'}
METHOD FB_exit : BOOL
VAR_INPUT
	(*  if TRUE, the exit method is called for exiting an instance that is copied afterwards (online change). *)
	bInCopyCode : BOOL;
END_VAR
END_METHOD

END_FUNCTION_BLOCK

// POUs/Motion/MC_Halt

{attribute 'c++_compatible'}
{attribute 'external_name' := 'MC_Halt_GUID_622541C0_FB19_1EA0_94E3_245323458AF0'}
{attribute 'TcIecLibraryType'}
{attribute 'hide_all_locals'}
(* 
		This function block commands a motion stop. The axis is transferred to the state DiscreteMotion, until
		zero dynamics is reached.
	 *)
FUNCTION_BLOCK MC_Halt
VAR_INPUT
	(* Reference to the axis *)
	{attribute 'GUID' := '71DDD02B-B842-4DDB-8CBB-D377B6714EDA'}
	{attribute 'Namespace' := 'Tc3_Mc3Ptp'}
	Axis : Type_SetValue1D;
	(* Trigger the command with rising edge *)
	Execute : BOOL;
END_VAR
VAR
	 {attribute 'hide'}
	_reserved1 : ARRAY [1..7] OF USINT;
END_VAR
VAR_INPUT
	(* Maximum deceleration ([PosUnit]/s^2, positive) *)
	Deceleration : LREAL := STRING_TO_LREAL('#Default');
	(* Maximum jerk ([PosUnit]/s^3, positive) *)
	Jerk : LREAL := STRING_TO_LREAL('#Default');
END_VAR
VAR
	 {attribute 'hide'}
	_reserved2 : UINT;
END_VAR
VAR_OUTPUT
	(* Zero dynamics has been reached, axis state is transferred to Standstill. *)
	Done : BOOL;
	(* Function block is not finished and new output values are to be expected *)
	Busy : BOOL;
	(* Function block has active control on the axis *)
	Active : BOOL;
	(* Command is aborted by another command *)
	CommandAborted : BOOL;
	(* Error occurred within function block *)
	Error : BOOL;
END_VAR
VAR
	 {attribute 'hide'}
	_reserved3 : USINT;
END_VAR
VAR_OUTPUT
	(* Error identifier *)
	ErrorId : UDINT;
END_VAR
VAR
	 {attribute 'hide'}
	_reserved4 : UINT_0_32;
	 {attribute 'hide'}
	_reserved5 : ARRAY [1..28] OF UINT_8_16;
	 {attribute 'hide'}
	_reserved6 : ARRAY [1..32] OF USINT;
END_VAR

{attribute 'TcTypeSystem'}

(* Internal method *)
{attribute 'hide'}
METHOD FB_init : BOOL
VAR_INPUT
	(*  if TRUE, the retain variables are initialized (warm start / cold start) *)
	bInitRetains : BOOL;
	(*  if TRUE, the instance afterwards gets moved into the copy code (online change) *)
	bInCopyCode : BOOL;
END_VAR
END_METHOD

{attribute 'TcTypeSystem'}

(* Internal method *)
{attribute 'hide'}
METHOD FB_exit : BOOL
VAR_INPUT
	(*  if TRUE, the exit method is called for exiting an instance that is copied afterwards (online change). *)
	bInCopyCode : BOOL;
END_VAR
END_METHOD

END_FUNCTION_BLOCK

// POUs/Motion/MC_GearInLegacy

{attribute 'c++_compatible'}
{attribute 'external_name' := 'MC_GearInLegacy_GUID_E97B502C_C319_1176_ABF8_971A701BCE43'}
{attribute 'TcIecLibraryType'}
{attribute 'hide_all_locals'}
{attribute 'hide'}
(* 
		This function block commands a ratio between the velocity of the slave and master axis.
	 *)
FUNCTION_BLOCK MC_GearInLegacy
VAR_INPUT
	(* Reference to the master axis *)
	{attribute 'GUID' := '67A81BB4-B31C-4E6F-99E0-6B37521E2266'}
	{attribute 'Namespace' := 'Tc3_Mc3Ptp'}
	Master : Type_ActValue1D;
	(* Reference to the slave axis *)
	{attribute 'GUID' := '71DDD02B-B842-4DDB-8CBB-D377B6714EDA'}
	{attribute 'Namespace' := 'Tc3_Mc3Ptp'}
	Slave : Type_SetValue1D;
	(* Trigger the command with rising edge *)
	Execute : BOOL;
END_VAR
VAR
	 {attribute 'hide'}
	_reserved1 : UINT_24_56;
END_VAR
VAR_INPUT
	(* Gear ratio numerator *)
	RatioNumerator : LREAL := 1.0;
	(* Gear ratio denominator *)
	RatioDenominator : UDINT := 1;
END_VAR
VAR
	 {attribute 'hide'}
	_reserved2 : UDINT;
END_VAR
VAR_INPUT
	(* Maximum slave velocity ([PosUnit]/s, positive) *)
	Velocity : LREAL := STRING_TO_LREAL('#Maximum');
	(* Maximum slave acceleration ([PosUnit]/s^2, positive) *)
	Acceleration : LREAL := STRING_TO_LREAL('#Default');
	(* Maximum slave deceleration ([PosUnit]/s^2, positive) *)
	Deceleration : LREAL := STRING_TO_LREAL('#Default');
	(* Maximum slave jerk ([PosUnit]/s^3, positive) *)
	Jerk : LREAL := STRING_TO_LREAL('#Default');
	(* Chronological sequence of the command *)
	{attribute 'Namespace' := 'Tc3_Mc3Base'}
	BufferMode : Tc3_Mc3Base.EBufferMode := Tc3_Mc3Base.EBufferMode.Aborting;
	(* Reaction if an error occurs in the master while this command is active *)
	{attribute 'Namespace' := 'Tc3_Mc3Base'}
	ReactionToMasterError : Tc3_Mc3Base.EReactionToMasterError := Tc3_Mc3Base.EReactionToMasterError.TriggerSlaveError;
	(* Reaction if an error occurs in the slave while this command is active *)
	{attribute 'Namespace' := 'Tc3_Mc3Base'}
	ReactionToSlaveError : Tc3_Mc3Base.EReactionToSlaveError := Tc3_Mc3Base.EReactionToSlaveError.TriggerMasterError;
	(* Advanced function block options *)
	{attribute 'hide'}
	{attribute 'GUID' := '62031914-E4A1-4C91-8071-51298070DBC2'}
	{attribute 'Namespace' := 'Tc3_Mc3Ptp'}
	Options : GearInLegacyOptions;
END_VAR
VAR_OUTPUT
	(* Synchronization established *)
	InGear : BOOL;
	(* Function block is not finished and new output values are to be expected *)
	Busy : BOOL;
	(* Function block has active control on the axis *)
	Active : BOOL;
	(* Command is aborted by another command *)
	CommandAborted : BOOL;
	(* Error occurred within function block *)
	Error : BOOL;
END_VAR
VAR
	 {attribute 'hide'}
	_reserved3 : USINT;
END_VAR
VAR_OUTPUT
	(* Error identifier *)
	ErrorId : UDINT;
	(* Master is in error state *)
	MasterHasError : BOOL;
END_VAR
VAR
	 {attribute 'hide'}
	_reserved4 : UINT_24_56;
	 {attribute 'hide'}
	_reserved5 : ARRAY [1..36] OF UINT_8_16;
	 {attribute 'hide'}
	_reserved6 : ARRAY [1..12] OF USINT;
END_VAR

{attribute 'TcTypeSystem'}

(* Internal method *)
{attribute 'hide'}
METHOD FB_init : BOOL
VAR_INPUT
	(*  if TRUE, the retain variables are initialized (warm start / cold start) *)
	bInitRetains : BOOL;
	(*  if TRUE, the instance afterwards gets moved into the copy code (online change) *)
	bInCopyCode : BOOL;
END_VAR
END_METHOD

{attribute 'TcTypeSystem'}

(* Internal method *)
{attribute 'hide'}
METHOD FB_exit : BOOL
VAR_INPUT
	(*  if TRUE, the exit method is called for exiting an instance that is copied afterwards (online change). *)
	bInCopyCode : BOOL;
END_VAR
END_METHOD

END_FUNCTION_BLOCK

// POUs/Motion/MC_GearInPosLegacy

{attribute 'c++_compatible'}
{attribute 'external_name' := 'MC_GearInPosLegacy_GUID_C97ACA83_50E9_16AC_98CB_727AB2F343E6'}
{attribute 'TcIecLibraryType'}
{attribute 'hide_all_locals'}
{attribute 'hide'}
(* 
		This function block commands a gear ratio between the position of the slave and master axes
		from the synchronization point onwards.
	 *)
FUNCTION_BLOCK MC_GearInPosLegacy
VAR_INPUT
	(* Reference to the master axis *)
	{attribute 'GUID' := '67A81BB4-B31C-4E6F-99E0-6B37521E2266'}
	{attribute 'Namespace' := 'Tc3_Mc3Ptp'}
	Master : Type_ActValue1D;
	(* Reference to the slave axis *)
	{attribute 'GUID' := '71DDD02B-B842-4DDB-8CBB-D377B6714EDA'}
	{attribute 'Namespace' := 'Tc3_Mc3Ptp'}
	Slave : Type_SetValue1D;
	(* Trigger the command with rising edge *)
	Execute : BOOL;
END_VAR
VAR
	 {attribute 'hide'}
	_reserved1 : UINT_24_56;
END_VAR
VAR_INPUT
	(* Gear ratio numerator *)
	RatioNumerator : LREAL := 1.0;
	(* Gear ratio denominator *)
	RatioDenominator : UDINT := 1;
END_VAR
VAR
	 {attribute 'hide'}
	_reserved2 : UDINT;
END_VAR
VAR_INPUT
	(* Position of master axis where master and slave axis are synchronized *)
	MasterSyncPosition : LREAL := STRING_TO_LREAL('#Invalid');
	(* Position of slave axis where master and slave axis are synchronized *)
	SlaveSyncPosition : LREAL := STRING_TO_LREAL('#Invalid');
	(* Maximum velocity during synchronization ([PosUnit]/s, positive) *)
	Velocity : LREAL := STRING_TO_LREAL('#Maximum');
	(* Maximum acceleration during synchronization ([PosUnit]/s^2, positive) *)
	Acceleration : LREAL := STRING_TO_LREAL('#Default');
	(* Maximum deceleration during synchronization ([PosUnit]/s^2, positive) *)
	Deceleration : LREAL := STRING_TO_LREAL('#Default');
	(* Maximum jerk during synchronization ([PosUnit]/s^3, positive) *)
	Jerk : LREAL := STRING_TO_LREAL('#Default');
	(* Chronological sequence of the command *)
	{attribute 'Namespace' := 'Tc3_Mc3Base'}
	BufferMode : Tc3_Mc3Base.EBufferMode := Tc3_Mc3Base.EBufferMode.Aborting;
	(* Reaction if an error occurs in the master while this command is active *)
	{attribute 'Namespace' := 'Tc3_Mc3Base'}
	ReactionToMasterError : Tc3_Mc3Base.EReactionToMasterError := Tc3_Mc3Base.EReactionToMasterError.TriggerSlaveError;
	(* Reaction if an error occurs in the slave while this command is active *)
	{attribute 'Namespace' := 'Tc3_Mc3Base'}
	ReactionToSlaveError : Tc3_Mc3Base.EReactionToSlaveError := Tc3_Mc3Base.EReactionToSlaveError.TriggerMasterError;
END_VAR
VAR
	 {attribute 'hide'}
	_reserved3 : UINT;
END_VAR
VAR_INPUT
	(* Advanced function block options *)
	{attribute 'hide'}
	{attribute 'GUID' := '64D35A59-CB0B-4CFE-AF1F-96B324BDF662'}
	{attribute 'Namespace' := 'Tc3_Mc3Ptp'}
	Options : GearInPosLegacyOptions;
END_VAR
VAR_OUTPUT
	(* Synchronization started *)
	{attribute 'hide'}
	StartSync : BOOL;
	(* Synchronization established *)
	InSync : BOOL;
	(* Function block is not finished and new output values are to be expected *)
	Busy : BOOL;
	(* Function block has active control on the axis *)
	Active : BOOL;
	(* Command is aborted by another command *)
	CommandAborted : BOOL;
	(* Error occurred within function block *)
	Error : BOOL;
END_VAR
VAR
	 {attribute 'hide'}
	_reserved4 : UINT;
END_VAR
VAR_OUTPUT
	(* Error identifier *)
	ErrorId : UDINT;
	(* Master is in error state *)
	MasterHasError : BOOL;
END_VAR
VAR
	 {attribute 'hide'}
	_reserved5 : UINT_24_56;
	 {attribute 'hide'}
	_reserved6 : ARRAY [1..28] OF UINT_8_16;
	 {attribute 'hide'}
	_reserved7 : ARRAY [1..28] OF USINT;
END_VAR

{attribute 'TcTypeSystem'}

(* Internal method *)
{attribute 'hide'}
METHOD FB_init : BOOL
VAR_INPUT
	(*  if TRUE, the retain variables are initialized (warm start / cold start) *)
	bInitRetains : BOOL;
	(*  if TRUE, the instance afterwards gets moved into the copy code (online change) *)
	bInCopyCode : BOOL;
END_VAR
END_METHOD

{attribute 'TcTypeSystem'}

(* Internal method *)
{attribute 'hide'}
METHOD FB_exit : BOOL
VAR_INPUT
	(*  if TRUE, the exit method is called for exiting an instance that is copied afterwards (online change). *)
	bInCopyCode : BOOL;
END_VAR
END_METHOD

END_FUNCTION_BLOCK

// POUs/Motion/MC_MoveAbsolute

{attribute 'c++_compatible'}
{attribute 'external_name' := 'MC_MoveAbsolute_GUID_920ED355_941C_193A_90B2_09B32FC4ED0F'}
{attribute 'TcIecLibraryType'}
{attribute 'hide_all_locals'}
(* 
		This function block commands a motion to a specified absolute position.
		Modulo parameters can be set in the options.
	 *)
FUNCTION_BLOCK MC_MoveAbsolute
VAR_INPUT
	(* Reference to the axis *)
	{attribute 'GUID' := '71DDD02B-B842-4DDB-8CBB-D377B6714EDA'}
	{attribute 'Namespace' := 'Tc3_Mc3Ptp'}
	Axis : Type_SetValue1D;
	(* Trigger the command with rising edge *)
	Execute : BOOL;
END_VAR
VAR
	 {attribute 'hide'}
	_reserved1 : ARRAY [1..7] OF USINT;
END_VAR
VAR_INPUT
	(* Commanded position ([PosUnit]) *)
	Position : LREAL := STRING_TO_LREAL('#Invalid');
	(* Maximum velocity ([PosUnit]/s, positive) *)
	Velocity : LREAL := STRING_TO_LREAL('#Invalid');
	(* Maximum acceleration ([PosUnit]/s^2, positive) *)
	Acceleration : LREAL := STRING_TO_LREAL('#Default');
	(* Maximum deceleration ([PosUnit]/s^2, positive) *)
	Deceleration : LREAL := STRING_TO_LREAL('#Default');
	(* Maximum jerk ([PosUnit]/s^3, positive) *)
	Jerk : LREAL := STRING_TO_LREAL('#Default');
	(* Chronological sequence of the command *)
	{attribute 'Namespace' := 'Tc3_Mc3Base'}
	BufferMode : Tc3_Mc3Base.EBufferMode := Tc3_Mc3Base.EBufferMode.Aborting;
END_VAR
VAR_OUTPUT
	(* Commanded position finally reached *)
	Done : BOOL;
	(* Function block is not finished and new output values are to be expected *)
	Busy : BOOL;
	(* Function block has active control on the axis *)
	Active : BOOL;
	(* Command is aborted by another command *)
	CommandAborted : BOOL;
	(* Error occurred within function block *)
	Error : BOOL;
END_VAR
VAR
	 {attribute 'hide'}
	_reserved2 : USINT;
END_VAR
VAR_OUTPUT
	(* Error identifier *)
	ErrorId : UDINT;
END_VAR
VAR
	 {attribute 'hide'}
	_reserved3 : UINT_0_32;
	 {attribute 'hide'}
	_reserved4 : ARRAY [1..36] OF UINT_8_16;
	 {attribute 'hide'}
	_reserved5 : ARRAY [1..16] OF USINT;
END_VAR

{attribute 'TcTypeSystem'}

(* Internal method *)
{attribute 'hide'}
METHOD FB_init : BOOL
VAR_INPUT
	(*  if TRUE, the retain variables are initialized (warm start / cold start) *)
	bInitRetains : BOOL;
	(*  if TRUE, the instance afterwards gets moved into the copy code (online change) *)
	bInCopyCode : BOOL;
END_VAR
END_METHOD

{attribute 'TcTypeSystem'}

(* Internal method *)
{attribute 'hide'}
METHOD FB_exit : BOOL
VAR_INPUT
	(*  if TRUE, the exit method is called for exiting an instance that is copied afterwards (online change). *)
	bInCopyCode : BOOL;
END_VAR
END_METHOD

END_FUNCTION_BLOCK

// POUs/Motion/MC_MoveModulo

{attribute 'c++_compatible'}
{attribute 'external_name' := 'MC_MoveModulo_GUID_79DD85B9_8F5D_1434_83CC_946C04F20F46'}
{attribute 'TcIecLibraryType'}
{attribute 'hide_all_locals'}
(* 
		This function block commands a motion to a specified modulo position.
	 *)
FUNCTION_BLOCK MC_MoveModulo
VAR_INPUT
	(* Reference to the axis *)
	{attribute 'GUID' := '71DDD02B-B842-4DDB-8CBB-D377B6714EDA'}
	{attribute 'Namespace' := 'Tc3_Mc3Ptp'}
	Axis : Type_SetValue1D;
	(* Trigger the command with rising edge *)
	Execute : BOOL;
END_VAR
VAR
	 {attribute 'hide'}
	_reserved1 : ARRAY [1..7] OF USINT;
END_VAR
VAR_INPUT
	(* Commanded modulo position ([PosUnit]) *)
	Position : LREAL := STRING_TO_LREAL('#Invalid');
	(* Number of additional modulo turns in the commanded direction. A value > 0 requires Direction <> EModuloDirection.ShortestDistance *)
	AdditionalTurns : UDINT := 0;
END_VAR
VAR
	 {attribute 'hide'}
	_reserved2 : UDINT;
END_VAR
VAR_INPUT
	(* Maximum velocity ([PosUnit]/s, positive) *)
	Velocity : LREAL := STRING_TO_LREAL('#Invalid');
	(* Maximum acceleration ([PosUnit]/s^2, positive) *)
	Acceleration : LREAL := STRING_TO_LREAL('#Default');
	(* Maximum deceleration ([PosUnit]/s^2, positive) *)
	Deceleration : LREAL := STRING_TO_LREAL('#Default');
	(* Maximum jerk ([PosUnit]/s^3, positive) *)
	Jerk : LREAL := STRING_TO_LREAL('#Default');
	(* Chronological sequence of the command *)
	{attribute 'Namespace' := 'Tc3_Mc3Base'}
	BufferMode : Tc3_Mc3Base.EBufferMode := Tc3_Mc3Base.EBufferMode.Aborting;
	(* Commanded direction. Must have value <> EModuloDirection.ShortestDistance if AdditionalTurns has value > 0. *)
	{attribute 'GUID' := '1798FE53-EDB6-4788-B12C-B2244F2AA2F6'}
	{attribute 'Namespace' := 'Tc3_Mc3Ptp'}
	Direction : EModuloDirection := EModuloDirection.ShortestDistance;
END_VAR
VAR_OUTPUT
	(* Commanded position finally reached *)
	Done : BOOL;
	(* Function block is not finished and new output values are to be expected *)
	Busy : BOOL;
	(* Function block has active control on the axis *)
	Active : BOOL;
	(* Command is aborted by another command *)
	CommandAborted : BOOL;
	(* Error occurred within function block *)
	Error : BOOL;
END_VAR
VAR
	 {attribute 'hide'}
	_reserved3 : ARRAY [1..3] OF USINT;
END_VAR
VAR_OUTPUT
	(* Error identifier *)
	ErrorId : UDINT;
END_VAR
VAR
	 {attribute 'hide'}
	_reserved4 : UINT_0_32;
	 {attribute 'hide'}
	_reserved5 : ARRAY [1..36] OF UINT_8_16;
	 {attribute 'hide'}
	_reserved6 : ARRAY [1..12] OF USINT;
END_VAR

{attribute 'TcTypeSystem'}

(* Internal method *)
{attribute 'hide'}
METHOD FB_init : BOOL
VAR_INPUT
	(*  if TRUE, the retain variables are initialized (warm start / cold start) *)
	bInitRetains : BOOL;
	(*  if TRUE, the instance afterwards gets moved into the copy code (online change) *)
	bInCopyCode : BOOL;
END_VAR
END_METHOD

{attribute 'TcTypeSystem'}

(* Internal method *)
{attribute 'hide'}
METHOD FB_exit : BOOL
VAR_INPUT
	(*  if TRUE, the exit method is called for exiting an instance that is copied afterwards (online change). *)
	bInCopyCode : BOOL;
END_VAR
END_METHOD

END_FUNCTION_BLOCK

// POUs/Motion/MC_MoveRelative

{attribute 'c++_compatible'}
{attribute 'external_name' := 'MC_MoveRelative_GUID_59B44DED_2369_1A00_A79B_5E5F05942967'}
{attribute 'TcIecLibraryType'}
{attribute 'hide_all_locals'}
(* 
		This function block commands a motion of a specified distance relative
		to the set position at the time the command gets active.
	 *)
FUNCTION_BLOCK MC_MoveRelative
VAR_INPUT
	(* Reference to the axis *)
	{attribute 'GUID' := '71DDD02B-B842-4DDB-8CBB-D377B6714EDA'}
	{attribute 'Namespace' := 'Tc3_Mc3Ptp'}
	Axis : Type_SetValue1D;
	(* Trigger the command with rising edge *)
	Execute : BOOL;
END_VAR
VAR
	 {attribute 'hide'}
	_reserved1 : ARRAY [1..7] OF USINT;
END_VAR
VAR_INPUT
	(* Relative distance ([PosUnit]) *)
	Distance : LREAL := STRING_TO_LREAL('#Invalid');
	(* Maximum velocity ([PosUnit]/s, positive) *)
	Velocity : LREAL := STRING_TO_LREAL('#Invalid');
	(* Maximum acceleration ([PosUnit]/s^2, positive) *)
	Acceleration : LREAL := STRING_TO_LREAL('#Default');
	(* Maximum deceleration ([PosUnit]/s^2, positive) *)
	Deceleration : LREAL := STRING_TO_LREAL('#Default');
	(* Maximum jerk ([PosUnit]/s^3, positive) *)
	Jerk : LREAL := STRING_TO_LREAL('#Default');
	(* Chronological sequence of the command *)
	{attribute 'Namespace' := 'Tc3_Mc3Base'}
	BufferMode : Tc3_Mc3Base.EBufferMode := Tc3_Mc3Base.EBufferMode.Aborting;
END_VAR
VAR_OUTPUT
	(* Commanded distance reached *)
	Done : BOOL;
	(* Function block is not finished and new output values are to be expected *)
	Busy : BOOL;
	(* Function block has active control on the axis *)
	Active : BOOL;
	(* Command is aborted by another command *)
	CommandAborted : BOOL;
	(* Error occurred within function block *)
	Error : BOOL;
END_VAR
VAR
	 {attribute 'hide'}
	_reserved2 : USINT;
END_VAR
VAR_OUTPUT
	(* Error identifier *)
	ErrorId : UDINT;
END_VAR
VAR
	 {attribute 'hide'}
	_reserved3 : UINT_0_32;
	 {attribute 'hide'}
	_reserved4 : ARRAY [1..28] OF UINT_8_16;
	 {attribute 'hide'}
	_reserved5 : ARRAY [1..32] OF USINT;
END_VAR

{attribute 'TcTypeSystem'}

(* Internal method *)
{attribute 'hide'}
METHOD FB_init : BOOL
VAR_INPUT
	(*  if TRUE, the retain variables are initialized (warm start / cold start) *)
	bInitRetains : BOOL;
	(*  if TRUE, the instance afterwards gets moved into the copy code (online change) *)
	bInCopyCode : BOOL;
END_VAR
END_METHOD

{attribute 'TcTypeSystem'}

(* Internal method *)
{attribute 'hide'}
METHOD FB_exit : BOOL
VAR_INPUT
	(*  if TRUE, the exit method is called for exiting an instance that is copied afterwards (online change). *)
	bInCopyCode : BOOL;
END_VAR
END_METHOD

END_FUNCTION_BLOCK

// POUs/Motion/MC_MoveVelocity

{attribute 'c++_compatible'}
{attribute 'external_name' := 'MC_MoveVelocity_GUID_38B7B259_5114_1519_AE61_5542A73A55A0'}
{attribute 'TcIecLibraryType'}
{attribute 'hide_all_locals'}
(* 
		This function block commands an endless movement with a specified velocity.
	 *)
FUNCTION_BLOCK MC_MoveVelocity
VAR_INPUT
	(* Reference to the axis *)
	{attribute 'GUID' := '71DDD02B-B842-4DDB-8CBB-D377B6714EDA'}
	{attribute 'Namespace' := 'Tc3_Mc3Ptp'}
	Axis : Type_SetValue1D;
	(* Trigger the command with rising edge *)
	Execute : BOOL;
END_VAR
VAR
	 {attribute 'hide'}
	_reserved1 : ARRAY [1..7] OF USINT;
END_VAR
VAR_INPUT
	(* Commanded velocity ([PosUnit]/s, the sign of this parameter determines the direction of movement) *)
	Velocity : LREAL := STRING_TO_LREAL('#Invalid');
	(* Maximum acceleration ([PosUnit]/s^2, positive) *)
	Acceleration : LREAL := STRING_TO_LREAL('#Default');
	(* Maximum deceleration ([PosUnit]/s^2, positive) *)
	Deceleration : LREAL := STRING_TO_LREAL('#Default');
	(* Maximum jerk ([PosUnit]/s^3, positive) *)
	Jerk : LREAL := STRING_TO_LREAL('#Default');
	(* Chronological sequence of the command *)
	{attribute 'Namespace' := 'Tc3_Mc3Base'}
	BufferMode : Tc3_Mc3Base.EBufferMode := Tc3_Mc3Base.EBufferMode.Aborting;
END_VAR
VAR_OUTPUT
	(* Commanded velocity reached *)
	InVelocity : BOOL;
	(* Function block is not finished and new output values are to be expected *)
	Busy : BOOL;
	(* Function block has active control on the axis *)
	Active : BOOL;
	(* Command is aborted by another command *)
	CommandAborted : BOOL;
	(* Error occurred within function block *)
	Error : BOOL;
END_VAR
VAR
	 {attribute 'hide'}
	_reserved2 : USINT;
END_VAR
VAR_OUTPUT
	(* Error identifier *)
	ErrorId : UDINT;
END_VAR
VAR
	 {attribute 'hide'}
	_reserved3 : UINT_0_32;
	 {attribute 'hide'}
	_reserved4 : ARRAY [1..12] OF UINT_8_16;
	 {attribute 'hide'}
	_reserved5 : ARRAY [1..64] OF USINT;
END_VAR

{attribute 'TcTypeSystem'}

(* Internal method *)
{attribute 'hide'}
METHOD FB_init : BOOL
VAR_INPUT
	(*  if TRUE, the retain variables are initialized (warm start / cold start) *)
	bInitRetains : BOOL;
	(*  if TRUE, the instance afterwards gets moved into the copy code (online change) *)
	bInCopyCode : BOOL;
END_VAR
END_METHOD

{attribute 'TcTypeSystem'}

(* Internal method *)
{attribute 'hide'}
METHOD FB_exit : BOOL
VAR_INPUT
	(*  if TRUE, the exit method is called for exiting an instance that is copied afterwards (online change). *)
	bInCopyCode : BOOL;
END_VAR
END_METHOD

END_FUNCTION_BLOCK

// POUs/Motion/MC_Stop

{attribute 'c++_compatible'}
{attribute 'external_name' := 'MC_Stop_GUID_94E328C9_775C_14D1_B2A8_713ACFD61F00'}
{attribute 'TcIecLibraryType'}
{attribute 'hide_all_locals'}
(* 
		This function block commands a motion stop and transfers the axis to the state Stopping.
		It aborts any ongoing function block execution. While the axis is in state Stopping, no other function block can
		perform any motion on the same axis. The Done output is set immediately after zero dynamics is reached.
		The axis remains in the state Stopping as long as Execute is TRUE or zero dynamics is not yet reached. As
		soon as Done is SET and Execute is FALSE the axis goes to state Standstill.
	 *)
FUNCTION_BLOCK MC_Stop
VAR_INPUT
	(* Reference to the axis *)
	{attribute 'GUID' := '71DDD02B-B842-4DDB-8CBB-D377B6714EDA'}
	{attribute 'Namespace' := 'Tc3_Mc3Ptp'}
	Axis : Type_SetValue1D;
	(* Trigger the command with rising edge. While this is TRUE, other function blocks will be rejected for the axis. *)
	Execute : BOOL;
END_VAR
VAR
	 {attribute 'hide'}
	_reserved1 : ARRAY [1..7] OF USINT;
END_VAR
VAR_INPUT
	(* Maximum deceleration ([PosUnit]/s^2, positive) *)
	Deceleration : LREAL := STRING_TO_LREAL('#Default');
	(* Maximum jerk ([PosUnit]/s^3, positive) *)
	Jerk : LREAL := STRING_TO_LREAL('#Default');
END_VAR
VAR_OUTPUT
	(* Zero dynamics has been reached *)
	Done : BOOL;
	(* Function block is not finished and new output values are to be expected *)
	Busy : BOOL;
	(* Function block has active control on the axis *)
	Active : BOOL;
	(* Command is aborted by another command *)
	CommandAborted : BOOL;
	(* Error occurred within function block *)
	Error : BOOL;
END_VAR
VAR
	 {attribute 'hide'}
	_reserved2 : ARRAY [1..3] OF USINT;
END_VAR
VAR_OUTPUT
	(* Error identifier *)
	ErrorId : UDINT;
END_VAR
VAR
	 {attribute 'hide'}
	_reserved3 : UINT_0_32;
	 {attribute 'hide'}
	_reserved4 : ARRAY [1..28] OF UINT_8_16;
	 {attribute 'hide'}
	_reserved5 : ARRAY [1..32] OF USINT;
END_VAR

{attribute 'TcTypeSystem'}

(* Internal method *)
{attribute 'hide'}
METHOD FB_init : BOOL
VAR_INPUT
	(*  if TRUE, the retain variables are initialized (warm start / cold start) *)
	bInitRetains : BOOL;
	(*  if TRUE, the instance afterwards gets moved into the copy code (online change) *)
	bInCopyCode : BOOL;
END_VAR
END_METHOD

{attribute 'TcTypeSystem'}

(* Internal method *)
{attribute 'hide'}
METHOD FB_exit : BOOL
VAR_INPUT
	(*  if TRUE, the exit method is called for exiting an instance that is copied afterwards (online change). *)
	bInCopyCode : BOOL;
END_VAR
END_METHOD

END_FUNCTION_BLOCK

// POUs/Motion/MC_Home

{attribute 'c++_compatible'}
{attribute 'external_name' := 'MC_Home_GUID_778DF838_FB0D_11F1_BE61_729CE3B81659'}
{attribute 'TcIecLibraryType'}
{attribute 'hide_all_locals'}
(* 
		This function block commands the axis to perform the 'search home' sequence.
	 *)
FUNCTION_BLOCK MC_Home
VAR_INPUT
	(* Reference to the axis *)
	{attribute 'GUID' := '71DDD02B-B842-4DDB-8CBB-D377B6714EDA'}
	{attribute 'Namespace' := 'Tc3_Mc3Ptp'}
	Axis : Type_SetValue1D;
	(* Trigger the command with rising edge *)
	Execute : BOOL;
END_VAR
VAR
	 {attribute 'hide'}
	_reserved1 : ARRAY [1..7] OF USINT;
END_VAR
VAR_INPUT
	(* Absolute position at the reference signal ([PosUnit]) *)
	Position : LREAL := STRING_TO_LREAL('#Default');
END_VAR
VAR_OUTPUT
	(* 'Search home' sequence succeeded *)
	Done : BOOL;
	(* Function block is not finished and new output values are to be expected *)
	Busy : BOOL;
	(* Function block has active control on the axis *)
	Active : BOOL;
	(* Command is aborted by another command *)
	CommandAborted : BOOL;
	(* Error occurred within function block *)
	Error : BOOL;
END_VAR
VAR
	 {attribute 'hide'}
	_reserved2 : ARRAY [1..3] OF USINT;
END_VAR
VAR_OUTPUT
	(* Error identifier *)
	ErrorId : UDINT;
END_VAR
VAR
	 {attribute 'hide'}
	_reserved3 : UINT_0_32;
	 {attribute 'hide'}
	_reserved4 : ARRAY [1..28] OF UINT_8_16;
	 {attribute 'hide'}
	_reserved5 : ARRAY [1..32] OF USINT;
END_VAR

{attribute 'TcTypeSystem'}

(* Internal method *)
{attribute 'hide'}
METHOD FB_init : BOOL
VAR_INPUT
	(*  if TRUE, the retain variables are initialized (warm start / cold start) *)
	bInitRetains : BOOL;
	(*  if TRUE, the instance afterwards gets moved into the copy code (online change) *)
	bInCopyCode : BOOL;
END_VAR
END_METHOD

{attribute 'TcTypeSystem'}

(* Internal method *)
{attribute 'hide'}
METHOD FB_exit : BOOL
VAR_INPUT
	(*  if TRUE, the exit method is called for exiting an instance that is copied afterwards (online change). *)
	bInCopyCode : BOOL;
END_VAR
END_METHOD

END_FUNCTION_BLOCK

// POUs/Motion/MC_Jog

{attribute 'c++_compatible'}
{attribute 'external_name' := 'MC_Jog_GUID_F8BFC424_4722_1591_9788_F166E691A525'}
{attribute 'TcIecLibraryType'}
{attribute 'hide_all_locals'}
(* 
		This function block enables an axis to be moved via manual keys in different modi.
	 *)
FUNCTION_BLOCK MC_Jog
VAR_INPUT
	(* Reference to the axis *)
	{attribute 'GUID' := '71DDD02B-B842-4DDB-8CBB-D377B6714EDA'}
	{attribute 'Namespace' := 'Tc3_Mc3Ptp'}
	Axis : Type_SetValue1D;
	(* The command is executed with a rising edge, and the axis is moved in positive direction.
		Depending on the mode, the axis moves as long as the signal remains TRUE, 
		or it stops automatically after a specified distance. *)
	JogForward : BOOL;
	(* The command is executed with a rising edge, and the axis is moved in negative direction.
		Depending on the mode, the axis moves as long as the signal remains TRUE, 
		or it stops automatically after a specified distance. *)
	JogBackward : BOOL;
	(* Determines the operation mode in which the manual function is executed. *)
	{attribute 'GUID' := '81AB5A5F-F1B6-4D6D-83FB-05EE8E17A103'}
	{attribute 'Namespace' := 'Tc3_Mc3Ptp'}
	Mode : EJogMode := EJogMode.StandardSlow;
END_VAR
VAR
	 {attribute 'hide'}
	_reserved1 : UDINT;
END_VAR
VAR_INPUT
	(* Distance for movements in Mode Inching  *)
	Distance : LREAL := STRING_TO_LREAL('#Ignore');
	(* Axis jog velocity parameter are used as default in case of operation modes StandardSlow and StandardFast. Otherwise Velocity has to be set. *)
	Velocity : LREAL := STRING_TO_LREAL('#Ignore');
	(* Maximum acceleration ([PosUnit]/s^2, positive) *)
	Acceleration : LREAL := STRING_TO_LREAL('#Default');
	(* Maximum deceleration ([PosUnit]/s^2, positive) *)
	Deceleration : LREAL := STRING_TO_LREAL('#Default');
	(* Maximum jerk ([PosUnit]/s^3, positive) *)
	Jerk : LREAL := STRING_TO_LREAL('#Default');
END_VAR
VAR_OUTPUT
	(* Function block has succeeded *)
	Done : BOOL;
	(* Function block is not finished and new output values are to be expected *)
	Busy : BOOL;
	(* Function block has active control on the axis *)
	Active : BOOL;
	(* Command is aborted by another command *)
	CommandAborted : BOOL;
	(* Error occurred within function block *)
	Error : BOOL;
END_VAR
VAR
	 {attribute 'hide'}
	_reserved2 : ARRAY [1..3] OF USINT;
END_VAR
VAR_OUTPUT
	(* Error identifier *)
	ErrorId : UDINT;
END_VAR
VAR
	 {attribute 'hide'}
	_reserved3 : UINT_0_32;
	 {attribute 'hide'}
	_reserved4 : ARRAY [1..116] OF UINT_8_16;
	 {attribute 'hide'}
	_reserved5 : ARRAY [1..336] OF USINT;
END_VAR

{attribute 'TcTypeSystem'}

(* Internal method *)
{attribute 'hide'}
METHOD FB_init : BOOL
VAR_INPUT
	(*  if TRUE, the retain variables are initialized (warm start / cold start) *)
	bInitRetains : BOOL;
	(*  if TRUE, the instance afterwards gets moved into the copy code (online change) *)
	bInCopyCode : BOOL;
END_VAR
END_METHOD

{attribute 'TcTypeSystem'}

(* Internal method *)
{attribute 'hide'}
METHOD FB_exit : BOOL
VAR_INPUT
	(*  if TRUE, the exit method is called for exiting an instance that is copied afterwards (online change). *)
	bInCopyCode : BOOL;
END_VAR
END_METHOD

END_FUNCTION_BLOCK

// POUs/Motion/MC_WaitForStableActualPosition

{attribute 'c++_compatible'}
{attribute 'external_name' := 'MC_WaitForStableActualPosition_GUID_395CBA62_FA8D_174D_A790_F2A6B953762B'}
{attribute 'TcIecLibraryType'}
{attribute 'hide_all_locals'}
(* 
		This function block waits for a stable actual position.
		It is always buffered and may only be triggered when the previous command ends with zero dynamics.
	 *)
FUNCTION_BLOCK MC_WaitForStableActualPosition
VAR_INPUT
	(* Reference to the axis *)
	{attribute 'GUID' := '67A81BB4-B31C-4E6F-99E0-6B37521E2266'}
	{attribute 'Namespace' := 'Tc3_Mc3Ptp'}
	Axis : Type_ActValue1D;
	(* Trigger the command with rising edge *)
	Execute : BOOL;
END_VAR
VAR
	 {attribute 'hide'}
	_reserved1 : ARRAY [1..7] OF USINT;
END_VAR
VAR_INPUT
	(* 
			Position tolerance around the set position ([PosUnit], positive). This defines the position window the actual position must be in in order to succeed.
		 *)
	PositionTolerance : LREAL := STRING_TO_LREAL('#Invalid');
	(* Duration (in seconds) that the actual position needs to consecutively stay inside the position window. Must have a value >= 0. *)
	WaitDuration : LREAL := STRING_TO_LREAL('#Invalid');
	(* 
			Duration (in seconds) after which an error is triggered if the actual position is not inside the position window.
			It can be left as 'Ignore' if no timeout is desired, otherwise must have a value > WaitDuration.
		 *)
	TimeoutDuration : LREAL := STRING_TO_LREAL('#Ignore');
END_VAR
VAR_OUTPUT
	(* Actual position is currently inside the position window. *)
	InPositionWindow : BOOL;
	(* Actual position has been consecutively inside the position window for at least WaitDuration. *)
	Done : BOOL;
	(* Function block is not finished and new output values are to be expected. *)
	Busy : BOOL;
	(* Function block has active control on the axis. 
		While Active is TRUE, the set position remains on the final position 
		of the previous command and the set dynamics remain zero. *)
	Active : BOOL;
	(* Command is aborted by another command. *)
	CommandAborted : BOOL;
	(* Error occurred within function block. *)
	Error : BOOL;
END_VAR
VAR
	 {attribute 'hide'}
	_reserved2 : UINT;
END_VAR
VAR_OUTPUT
	(* Error identifier *)
	ErrorId : UDINT;
END_VAR
VAR
	 {attribute 'hide'}
	_reserved3 : UINT_0_32;
	 {attribute 'hide'}
	_reserved4 : ARRAY [1..28] OF UINT_8_16;
	 {attribute 'hide'}
	_reserved5 : ARRAY [1..32] OF USINT;
END_VAR

{attribute 'TcTypeSystem'}

(* Internal method *)
{attribute 'hide'}
METHOD FB_init : BOOL
VAR_INPUT
	(*  if TRUE, the retain variables are initialized (warm start / cold start) *)
	bInitRetains : BOOL;
	(*  if TRUE, the instance afterwards gets moved into the copy code (online change) *)
	bInCopyCode : BOOL;
END_VAR
END_METHOD

{attribute 'TcTypeSystem'}

(* Internal method *)
{attribute 'hide'}
METHOD FB_exit : BOOL
VAR_INPUT
	(*  if TRUE, the exit method is called for exiting an instance that is copied afterwards (online change). *)
	bInCopyCode : BOOL;
END_VAR
END_METHOD

END_FUNCTION_BLOCK

// POUs/Motion/MC_PhasingAbsolute

{attribute 'c++_compatible'}
{attribute 'external_name' := 'MC_PhasingAbsolute_GUID_EA7E8009_70F8_1952_A489_35241184855D'}
{attribute 'TcIecLibraryType'}
{attribute 'hide_all_locals'}
(* 
		This function block commands an absolute phase shift in the master position of a synchronized slave axis.
		It is only valid for camming synchronization. The master axis is not aware of the phase shift.
	 *)
FUNCTION_BLOCK MC_PhasingAbsolute
VAR_INPUT
	(* Reference to the master axis *)
	{attribute 'GUID' := '67A81BB4-B31C-4E6F-99E0-6B37521E2266'}
	{attribute 'Namespace' := 'Tc3_Mc3Ptp'}
	Master : Type_ActValue1D;
	(* Reference to the slave axis *)
	{attribute 'GUID' := '71DDD02B-B842-4DDB-8CBB-D377B6714EDA'}
	{attribute 'Namespace' := 'Tc3_Mc3Ptp'}
	Slave : Type_SetValue1D;
	(* Trigger the command with rising edge *)
	Execute : BOOL;
END_VAR
VAR
	 {attribute 'hide'}
	_reserved1 : UINT_24_56;
END_VAR
VAR_INPUT
	(* Absolute phase difference in master position of the slave axis ([PosUnit]) *)
	PhaseShift : LREAL := STRING_TO_LREAL('#Invalid');
	(* Maximum velocity ([PosUnit]/s, positive) *)
	Velocity : LREAL := STRING_TO_LREAL('#Invalid');
	(* Maximum acceleration ([PosUnit]/s^2, positive) *)
	Acceleration : LREAL := STRING_TO_LREAL('#Invalid');
	(* Maximum deceleration ([PosUnit]/s^2, positive) *)
	Deceleration : LREAL := STRING_TO_LREAL('#Invalid');
	(* Maximum jerk ([PosUnit]/s^3, positive) *)
	Jerk : LREAL := STRING_TO_LREAL('#Invalid');
END_VAR
VAR_OUTPUT
	(* Commanded phasing reached *)
	Done : BOOL;
	(* Function block is not finished and new output values are to be expected *)
	Busy : BOOL;
	(* Function block has active control on the axis *)
	Active : BOOL;
	(* Command is aborted by another command *)
	CommandAborted : BOOL;
	(* Error occurred within function block *)
	Error : BOOL;
END_VAR
VAR
	 {attribute 'hide'}
	_reserved2 : ARRAY [1..3] OF USINT;
END_VAR
VAR_OUTPUT
	(* Error identifier *)
	ErrorId : UDINT;
END_VAR
VAR
	 {attribute 'hide'}
	_reserved3 : UDINT;
END_VAR
VAR_OUTPUT
	AbsolutePhaseShift : LREAL;
END_VAR
VAR
	 {attribute 'hide'}
	_reserved4 : UINT_0_32;
	 {attribute 'hide'}
	_reserved5 : ARRAY [1..36] OF UINT_8_16;
	 {attribute 'hide'}
	_reserved6 : ARRAY [1..12] OF USINT;
END_VAR

{attribute 'TcTypeSystem'}

(* Internal method *)
{attribute 'hide'}
METHOD FB_init : BOOL
VAR_INPUT
	(*  if TRUE, the retain variables are initialized (warm start / cold start) *)
	bInitRetains : BOOL;
	(*  if TRUE, the instance afterwards gets moved into the copy code (online change) *)
	bInCopyCode : BOOL;
END_VAR
END_METHOD

{attribute 'TcTypeSystem'}

(* Internal method *)
{attribute 'hide'}
METHOD FB_exit : BOOL
VAR_INPUT
	(*  if TRUE, the exit method is called for exiting an instance that is copied afterwards (online change). *)
	bInCopyCode : BOOL;
END_VAR
END_METHOD

END_FUNCTION_BLOCK

// POUs/Motion/MC_PhasingRelative

{attribute 'c++_compatible'}
{attribute 'external_name' := 'MC_PhasingRelative_GUID_F11F065F_B087_1FD0_AD03_4BE9CCC19A83'}
{attribute 'TcIecLibraryType'}
{attribute 'hide_all_locals'}
(* 
		This function block commands a relative phase shift in the master position of a synchronized slave axis.
		It is only valid for camming synchronization. The master axis is not aware of the phase shift.
	 *)
FUNCTION_BLOCK MC_PhasingRelative
VAR_INPUT
	(* Reference to the master axis *)
	{attribute 'GUID' := '67A81BB4-B31C-4E6F-99E0-6B37521E2266'}
	{attribute 'Namespace' := 'Tc3_Mc3Ptp'}
	Master : Type_ActValue1D;
	(* Reference to the slave axis *)
	{attribute 'GUID' := '71DDD02B-B842-4DDB-8CBB-D377B6714EDA'}
	{attribute 'Namespace' := 'Tc3_Mc3Ptp'}
	Slave : Type_SetValue1D;
	(* Trigger the command with rising edge *)
	Execute : BOOL;
END_VAR
VAR
	 {attribute 'hide'}
	_reserved1 : UINT_24_56;
END_VAR
VAR_INPUT
	(* Additional phase difference in master position of the slave axis ([PosUnit]) *)
	PhaseShift : LREAL := STRING_TO_LREAL('#Invalid');
	(* Maximum velocity ([PosUnit]/s, positive) *)
	Velocity : LREAL := STRING_TO_LREAL('#Invalid');
	(* Maximum acceleration ([PosUnit]/s^2, positive) *)
	Acceleration : LREAL := STRING_TO_LREAL('#Invalid');
	(* Maximum deceleration ([PosUnit]/s^2, positive) *)
	Deceleration : LREAL := STRING_TO_LREAL('#Invalid');
	(* Maximum jerk ([PosUnit]/s^3, positive) *)
	Jerk : LREAL := STRING_TO_LREAL('#Invalid');
END_VAR
VAR_OUTPUT
	(* Commanded phasing reached *)
	Done : BOOL;
	(* Function Block is not finished and new output values are to be expected *)
	Busy : BOOL;
	(* Function block has active control on the axis *)
	Active : BOOL;
	(* Command is aborted by another command *)
	CommandAborted : BOOL;
	(* Error occurred within function block *)
	Error : BOOL;
END_VAR
VAR
	 {attribute 'hide'}
	_reserved2 : ARRAY [1..3] OF USINT;
END_VAR
VAR_OUTPUT
	(* Error identifier *)
	ErrorId : UDINT;
END_VAR
VAR
	 {attribute 'hide'}
	_reserved3 : UDINT;
END_VAR
VAR_OUTPUT
	CoveredPhaseShift : LREAL;
END_VAR
VAR
	 {attribute 'hide'}
	_reserved4 : UINT_0_32;
	 {attribute 'hide'}
	_reserved5 : ARRAY [1..36] OF UINT_8_16;
	 {attribute 'hide'}
	_reserved6 : ARRAY [1..12] OF USINT;
END_VAR

{attribute 'TcTypeSystem'}

(* Internal method *)
{attribute 'hide'}
METHOD FB_init : BOOL
VAR_INPUT
	(*  if TRUE, the retain variables are initialized (warm start / cold start) *)
	bInitRetains : BOOL;
	(*  if TRUE, the instance afterwards gets moved into the copy code (online change) *)
	bInCopyCode : BOOL;
END_VAR
END_METHOD

{attribute 'TcTypeSystem'}

(* Internal method *)
{attribute 'hide'}
METHOD FB_exit : BOOL
VAR_INPUT
	(*  if TRUE, the exit method is called for exiting an instance that is copied afterwards (online change). *)
	bInCopyCode : BOOL;
END_VAR
END_METHOD

END_FUNCTION_BLOCK

// POUs/Motion/MC_HaltPhasing

{attribute 'c++_compatible'}
{attribute 'external_name' := 'MC_HaltPhasing_GUID_33DF456A_9802_1C72_890A_D2020DFCE950'}
{attribute 'TcIecLibraryType'}
{attribute 'hide_all_locals'}
(* 
		This function block commands a phase shift stop in the master position of a synchronized slave axis.
		It is only valid for camming synchronization. The master axis is not aware of the phase shift.
	 *)
FUNCTION_BLOCK MC_HaltPhasing
VAR_INPUT
	(* Reference to the master axis *)
	{attribute 'GUID' := '67A81BB4-B31C-4E6F-99E0-6B37521E2266'}
	{attribute 'Namespace' := 'Tc3_Mc3Ptp'}
	Master : Type_ActValue1D;
	(* Reference to the slave axis *)
	{attribute 'GUID' := '71DDD02B-B842-4DDB-8CBB-D377B6714EDA'}
	{attribute 'Namespace' := 'Tc3_Mc3Ptp'}
	Slave : Type_SetValue1D;
	(* Trigger the command with rising edge *)
	Execute : BOOL;
END_VAR
VAR
	 {attribute 'hide'}
	_reserved1 : UINT_24_56;
END_VAR
VAR_INPUT
	(* Maximum deceleration ([PosUnit]/s^2, positive) *)
	Deceleration : LREAL := STRING_TO_LREAL('#Invalid');
	(* Maximum jerk ([PosUnit]/s^3, positive) *)
	Jerk : LREAL := STRING_TO_LREAL('#Invalid');
END_VAR
VAR_OUTPUT
	(* Zero dynamics has been reached, axis state is transferred to Standstill. *)
	Done : BOOL;
	(* Function block is not finished and new output values are to be expected *)
	Busy : BOOL;
	(* Function block has active control on the axis *)
	Active : BOOL;
	(* Command is aborted by another command *)
	CommandAborted : BOOL;
	(* Error occurred within function block *)
	Error : BOOL;
END_VAR
VAR
	 {attribute 'hide'}
	_reserved2 : ARRAY [1..3] OF USINT;
END_VAR
VAR_OUTPUT
	(* Error identifier *)
	ErrorId : UDINT;
END_VAR
VAR
	 {attribute 'hide'}
	_reserved3 : UINT_0_32;
	 {attribute 'hide'}
	_reserved4 : ARRAY [1..36] OF UINT_8_16;
	 {attribute 'hide'}
	_reserved5 : ARRAY [1..16] OF USINT;
END_VAR

{attribute 'TcTypeSystem'}

(* Internal method *)
{attribute 'hide'}
METHOD FB_init : BOOL
VAR_INPUT
	(*  if TRUE, the retain variables are initialized (warm start / cold start) *)
	bInitRetains : BOOL;
	(*  if TRUE, the instance afterwards gets moved into the copy code (online change) *)
	bInCopyCode : BOOL;
END_VAR
END_METHOD

{attribute 'TcTypeSystem'}

(* Internal method *)
{attribute 'hide'}
METHOD FB_exit : BOOL
VAR_INPUT
	(*  if TRUE, the exit method is called for exiting an instance that is copied afterwards (online change). *)
	bInCopyCode : BOOL;
END_VAR
END_METHOD

END_FUNCTION_BLOCK
